ABB RobotStudio station: Celda_Robotica_Pintura_APM.rspag

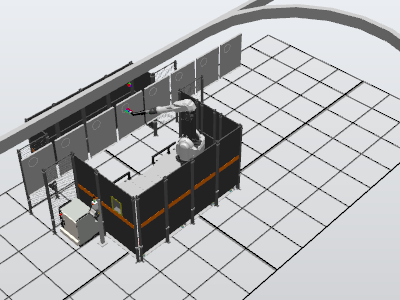
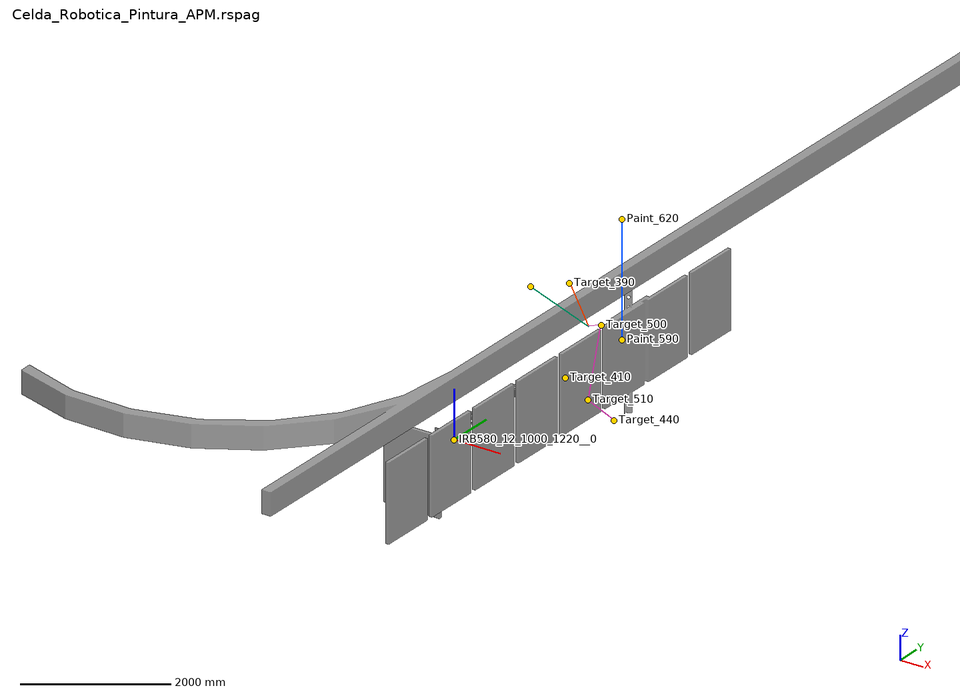
[picture v1: parts stored in the station drawn from their meshes, with robot base, taught points and paths (robot models come from the ABB library and are not in the file)]
--- station ---
Station Celda_Robotica_2_APM (saved by RobotStudio 23.3.10550.0)
Controller Controlador_Pintura_v2, task T_ROB1: task frame (RAPID world) sits at (2600, 704.38, 2665.12) mm, rotated rx 180 ry 0 rz 90 deg in the station
Controller Controlador_Pintura_v2
  mechanical unit ROB_1: IRB580_12_1000_1220__01, 6 joints, base frame (-1683.63, -1674.53, 2052.21) mm, rotated rx 180 ry 0 rz 0 deg
  mechanical unit CNV1: ?, 1 joints, base frame (-1079.32, 0, 0) mm
Layout (positions relative to the parent item):
  - Fence_800_AW [part, from Libraries\f3bba005-ce8c-4d92-bad9-ebedfeb7daa5fence_800_aw.rslib] at (-415.23, -1488.01, 0) mm
  - Pedestal_h440 [part, from Libraries\Pedestal_h440.rslib] at (891.47, -950, 628.29) mm, rotated rx 0 ry 0 rz 90 deg
  - sPallet250R_Single_rev1 [part, from Libraries\sPallet250R_Single_rev1.rslib] at (0, 1.5, 0) mm
  - ROBOBEL926_T_TD_03 [mechanism, from Libraries\ROBOBEL926_T_TD_03.rslib] at (1986.48, -515.02, 1892.16) mm, rotated rx -89.96 ry 0.02 rz -29.27 deg
  - Fence_800 [part, from Libraries\f3bba005-ce8c-4d92-bad9-ebedfeb7daa5fence_800_aw.rslib] at (-415.23, 1208.98, 0) mm
  - Fence_800_2 [part, from Libraries\f3bba005-ce8c-4d92-bad9-ebedfeb7daa5fence_800_aw.rslib] at (-415.23, -588.05, 0) mm
  - Fence_800_3 [part, from Libraries\f3bba005-ce8c-4d92-bad9-ebedfeb7daa5fence_800_aw.rslib] at (-415.23, 310.24, 0) mm
  - Fence_800_4 [part, from Libraries\f3bba005-ce8c-4d92-bad9-ebedfeb7daa5fence_800_aw.rslib] at (1805.95, -1488.01, 0) mm, rotated rx 0 ry 0 rz 90 deg
  - Fence_800_5 [part, from Libraries\f3bba005-ce8c-4d92-bad9-ebedfeb7daa5fence_800_aw.rslib] at (495.14, -1488.01, 0) mm, rotated rx 0 ry 0 rz 90 deg
  - Fence_800_6 [part, from Libraries\f3bba005-ce8c-4d92-bad9-ebedfeb7daa5fence_800_aw.rslib] at (1133.79, -1488.01, 0) mm, rotated rx 0 ry 0 rz 90 deg
  - Fence_800_7 [part, from Libraries\f3bba005-ce8c-4d92-bad9-ebedfeb7daa5fence_800_aw.rslib] at (2834.37, 2145.85, 0) mm, rotated rx 0 ry 0 rz -90 deg
  - IRC5_Singel-Cabinet [part, from Libraries\IRC5_Singel-Cabinet.rslib] at (1354.6, 2720.15, 100) mm, rotated rx 90 ry 0 rz 180 deg
  - Operator_panel [part, from Libraries\Operator_panel.rslib] at (714, 2359.02, 0) mm, rotated rx 0 ry 0 rz 90 deg
  - MeshModel_BoundingBox [graphiccomponentgroup]
  - MeshModel_ClippingPlane [graphiccomponentgroup]
  - MeshModel_ClippingCurve [graphiccomponentgroup]
  - Part5 [part], size 130 x 63 x 230 mm
  - Part6 [part], size 100 x 10 x 140 mm
  - Part7 [part], size 150 x 1 x 250 mm
  - Part8 [graphiccomponentgroup] at (0, 0, 420.53) mm
    - Part8_1 [part] at (2372.99, 892.19, 255.6) mm, rotated rx 90 ry 0 rz -151.74 deg, size 8 x 8 x 3 mm
    - Part8_2 [part] at (2372.99, 892.19, 255.6) mm, rotated rx 90 ry 0 rz -151.74 deg, size 8 x 8 x 3 mm
    - Part8_3 [part] at (2372.99, 892.19, 255.6) mm, rotated rx 90 ry 0 rz -151.74 deg, size 50 x 50 x 3 mm
    - Part8_4 [part] at (2372.99, 892.19, 255.6) mm, rotated rx 90 ry 0 rz -151.74 deg, size 8 x 8 x 3 mm
    - Part8_5 [part] at (2372.99, 892.19, 255.6) mm, rotated rx 90 ry 0 rz -151.74 deg, size 8 x 8 x 3 mm
    - Part8_6 [part] at (2372.99, 892.19, 255.6) mm, rotated rx 90 ry 0 rz -151.74 deg, size 50 x 50 x 3 mm
    - Part8_7 [part] at (2372.99, 892.19, 255.6) mm, rotated rx 90 ry 0 rz -151.74 deg, size 8 x 8 x 3 mm
    - Part8_8 [part] at (2372.99, 892.19, 255.6) mm, rotated rx 90 ry 0 rz -151.74 deg, size 50 x 50 x 3 mm
    - Part8_9 [part] at (2372.99, 892.19, 255.6) mm, rotated rx 90 ry 0 rz -151.74 deg, size 8 x 8 x 3 mm
    - Part8_10 [part] at (2372.99, 892.19, 255.6) mm, rotated rx 90 ry 0 rz -151.74 deg, size 50 x 50 x 3 mm
    - Part8_11 [part] at (2372.99, 892.19, 255.6) mm, rotated rx 90 ry 0 rz -151.74 deg, size 50 x 50 x 3 mm
    - Part8_12 [part] at (2372.99, 892.19, 255.6) mm, rotated rx 90 ry 0 rz -151.74 deg, size 8 x 8 x 3 mm
    - Part8_13 [part] at (2372.99, 892.19, 255.6) mm, rotated rx 90 ry 0 rz -151.74 deg, size 50 x 50 x 3 mm
    - Part8_14 [part] at (2372.99, 892.19, 255.6) mm, rotated rx 90 ry 0 rz -151.74 deg, size 50 x 50 x 3 mm
    - Part8_15 [part] at (2372.99, 892.19, 255.6) mm, rotated rx 90 ry 0 rz -151.74 deg, size 8 x 8 x 3 mm
    - Part8_16 [part] at (2372.99, 892.19, 255.6) mm, rotated rx 90 ry 0 rz -151.74 deg, size 50 x 50 x 3 mm
    - Part8_17 [part] at (2372.99, 892.19, 255.6) mm, rotated rx 90 ry 0 rz -151.74 deg, size 8 x 8 x 3 mm
    - Part8_18 [part] at (2372.99, 892.19, 255.6) mm, rotated rx 90 ry 0 rz -151.74 deg, size 50 x 50 x 3 mm
    - Part8_19 [part] at (2372.99, 892.19, 255.6) mm, rotated rx 90 ry 0 rz -151.74 deg, size 50 x 50 x 3 mm
    - Part8_20 [part] at (2372.99, 892.19, 255.6) mm, rotated rx 90 ry 0 rz -151.74 deg, size 8 x 8 x 3 mm
    - Part8_21 [part] at (2372.99, 892.19, 255.6) mm, rotated rx 90 ry 0 rz -151.74 deg, size 50 x 50 x 3 mm
    - Part8_22 [part] at (2372.99, 892.19, 255.6) mm, rotated rx 90 ry 0 rz -151.74 deg, size 50 x 50 x 3 mm
    - Part8_23 [part] at (2372.99, 892.19, 255.6) mm, rotated rx 90 ry 0 rz -151.74 deg, size 50 x 50 x 3 mm
    - Part8_24 [part] at (2372.99, 892.19, 255.6) mm, rotated rx 90 ry 0 rz -151.74 deg, size 8 x 8 x 3 mm
    - Part8_25 [part] at (2372.99, 892.19, 255.6) mm, rotated rx 90 ry 0 rz -151.74 deg, size 8 x 8 x 3 mm
    - Part8_26 [part] at (2372.99, 892.19, 255.6) mm, rotated rx 90 ry 0 rz -151.74 deg, size 50 x 50 x 3 mm
    - Part8_27 [part] at (2372.99, 892.19, 255.6) mm, rotated rx 90 ry 0 rz -151.74 deg, size 8 x 8 x 3 mm
    - Part8_28 [part] at (2372.99, 892.19, 255.6) mm, rotated rx 90 ry 0 rz -151.74 deg, size 8 x 8 x 3 mm
    - Part8_29 [part] at (2372.99, 892.19, 255.6) mm, rotated rx 90 ry 0 rz -151.74 deg, size 50 x 50 x 3 mm
    - Part8_30 [part] at (2372.99, 892.19, 255.6) mm, rotated rx 90 ry 0 rz -151.74 deg, size 8 x 8 x 3 mm
    - Part8_31 [part] at (2372.99, 892.19, 255.6) mm, rotated rx 90 ry 0 rz -151.74 deg, size 3 x 8 x 8 mm
    - Part8_32 [part] at (2372.99, 892.19, 255.6) mm, rotated rx 90 ry 0 rz -151.74 deg, size 3 x 8 x 8 mm
    - Part8_33 [part] at (2372.99, 892.19, 255.6) mm, rotated rx 90 ry 0 rz -151.74 deg, size 3 x 50 x 50 mm
    - Part8_34 [part] at (2372.99, 892.19, 255.6) mm, rotated rx 90 ry 0 rz -151.74 deg, size 3 x 8 x 8 mm
    - Part8_35 [part] at (2372.99, 892.19, 255.6) mm, rotated rx 90 ry 0 rz -151.74 deg, size 3 x 8 x 8 mm
    - Part8_36 [part] at (2372.99, 892.19, 255.6) mm, rotated rx 90 ry 0 rz -151.74 deg, size 3 x 50 x 50 mm
    - Part8_37 [part] at (2372.99, 892.19, 255.6) mm, rotated rx 90 ry 0 rz -151.74 deg, size 3 x 8 x 8 mm
    - Part8_38 [part] at (2372.99, 892.19, 255.6) mm, rotated rx 90 ry 0 rz -151.74 deg, size 3 x 50 x 50 mm
    - Part8_39 [part] at (2372.99, 892.19, 255.6) mm, rotated rx 90 ry 0 rz -151.74 deg, size 3 x 8 x 8 mm
    - Part8_40 [part] at (2372.99, 892.19, 255.6) mm, rotated rx 90 ry 0 rz -151.74 deg, size 3 x 50 x 50 mm
    - Part8_41 [part] at (2372.99, 892.19, 255.6) mm, rotated rx 90 ry 0 rz -151.74 deg, size 3 x 50 x 50 mm
    - Part8_42 [part] at (2372.99, 892.19, 255.6) mm, rotated rx 90 ry 0 rz -151.74 deg, size 3 x 8 x 8 mm
    - Part8_43 [part] at (2372.99, 892.19, 255.6) mm, rotated rx 90 ry 0 rz -151.74 deg, size 3 x 50 x 50 mm
    - Part8_44 [part] at (2372.99, 892.19, 255.6) mm, rotated rx 90 ry 0 rz -151.74 deg, size 3 x 50 x 50 mm
    - Part8_45 [part] at (2372.99, 892.19, 255.6) mm, rotated rx 90 ry 0 rz -151.74 deg, size 3 x 8 x 8 mm
    - Part8_46 [part] at (2372.99, 892.19, 255.6) mm, rotated rx 90 ry 0 rz -151.74 deg, size 3 x 50 x 50 mm
    - Part8_47 [part] at (2372.99, 892.19, 255.6) mm, rotated rx 90 ry 0 rz -151.74 deg, size 3 x 8 x 8 mm
    - Part8_48 [part] at (2372.99, 892.19, 255.6) mm, rotated rx 90 ry 0 rz -151.74 deg, size 3 x 50 x 50 mm
    - Part8_49 [part] at (2372.99, 892.19, 255.6) mm, rotated rx 90 ry 0 rz -151.74 deg, size 3 x 50 x 50 mm
    - Part8_50 [part] at (2372.99, 892.19, 255.6) mm, rotated rx 90 ry 0 rz -151.74 deg, size 3 x 8 x 8 mm
    - Part8_51 [part] at (2372.99, 892.19, 255.6) mm, rotated rx 90 ry 0 rz -151.74 deg, size 3 x 50 x 50 mm
    - Part8_52 [part] at (2372.99, 892.19, 255.6) mm, rotated rx 90 ry 0 rz -151.74 deg, size 3 x 50 x 50 mm
    - Part8_53 [part] at (2372.99, 892.19, 255.6) mm, rotated rx 90 ry 0 rz -151.74 deg, size 3 x 50 x 50 mm
    - Part8_54 [part] at (2372.99, 892.19, 255.6) mm, rotated rx 90 ry 0 rz -151.74 deg, size 3 x 8 x 8 mm
    - Part8_55 [part] at (2372.99, 892.19, 255.6) mm, rotated rx 90 ry 0 rz -151.74 deg, size 3 x 8 x 8 mm
    - Part8_56 [part] at (2372.99, 892.19, 255.6) mm, rotated rx 90 ry 0 rz -151.74 deg, size 3 x 50 x 50 mm
    - Part8_57 [part] at (2372.99, 892.19, 255.6) mm, rotated rx 90 ry 0 rz -151.74 deg, size 3 x 8 x 8 mm
    - Part8_58 [part] at (2372.99, 892.19, 255.6) mm, rotated rx 90 ry 0 rz -151.74 deg, size 3 x 8 x 8 mm
    - Part8_59 [part] at (2372.99, 892.19, 255.6) mm, rotated rx 90 ry 0 rz -151.74 deg, size 3 x 50 x 50 mm
    - Part8_60 [part] at (2372.99, 892.19, 255.6) mm, rotated rx 90 ry 0 rz -151.74 deg, size 3 x 8 x 8 mm
    - Part8_61 [part] at (2372.99, 892.19, 255.6) mm, rotated rx 90 ry 0 rz -151.74 deg, size 100 x 2000 x 0 mm
    - Part8_62 [part] at (2372.99, 892.19, 255.6) mm, rotated rx 90 ry 0 rz -151.74 deg, size 0 x 2000 x 3 mm
    - Part8_63 [part] at (2372.99, 892.19, 255.6) mm, rotated rx 90 ry 0 rz -151.74 deg, size 97 x 2000 x 0 mm
    - Part8_64 [part] at (2372.99, 892.19, 255.6) mm, rotated rx 90 ry 0 rz -151.74 deg, size 0 x 2000 x 97 mm
    - Part8_65 [part] at (2372.99, 892.19, 255.6) mm, rotated rx 90 ry 0 rz -151.74 deg, size 3 x 2000 x 0 mm
    - Part8_66 [part] at (2372.99, 892.19, 255.6) mm, rotated rx 90 ry 0 rz -151.74 deg, size 0 x 2000 x 100 mm
    - Part8_67 [part] at (2372.99, 892.19, 255.6) mm, rotated rx 90 ry 0 rz -151.74 deg, size 100 x 0 x 100 mm
    - Part8_68 [part] at (2372.99, 892.19, 255.6) mm, rotated rx 90 ry 0 rz -151.74 deg, size 100 x 0 x 100 mm
  - Fence_800_8 [part, from Libraries\f3bba005-ce8c-4d92-bad9-ebedfeb7daa5fence_800_aw.rslib] at (927.36, 2145.85, 0) mm, rotated rx 0 ry 0 rz -90 deg
  - Fence_800_9 [part, from Libraries\f3bba005-ce8c-4d92-bad9-ebedfeb7daa5fence_800_aw.rslib] at (3699.9, 2145.85, 0) mm, rotated rx 0 ry 0 rz 180 deg
  - Fence_1200_AW [part, from Libraries\48bacffd-50a7-42ca-88af-306811f71c63fence_1200_aw_ts.rslib] at (-372.93, 2145.84, -3.07) mm, rotated rx 0 ry 0 rz -90 deg
  - Fence_800_10 [part, from Libraries\f3bba005-ce8c-4d92-bad9-ebedfeb7daa5fence_800_aw.rslib] at (3699.9, 1245.66, 0) mm, rotated rx 0 ry 0 rz 180 deg
  - Fence_800_11 [part, from Libraries\f3bba005-ce8c-4d92-bad9-ebedfeb7daa5fence_800_aw.rslib] at (3699.9, 346.45, 0) mm, rotated rx 0 ry 0 rz 180 deg
  - Fence_800_12 [part, from Libraries\f3bba005-ce8c-4d92-bad9-ebedfeb7daa5fence_800_aw.rslib] at (3699.9, -552.32, 0) mm, rotated rx 0 ry 0 rz 180 deg
  - Fence_800_13 [part, from Libraries\f3bba005-ce8c-4d92-bad9-ebedfeb7daa5fence_800_aw.rslib] at (3709.4, -1462.88, 0) mm, rotated rx 0 ry 0 rz 90 deg
  - Troax_800_Poles [part, from Libraries\9d9a1cc8-97d7-4a8c-92c3-0b58d3e22f0ctroax_800_poles.rslib] at (1795.44, -1936.07, 0) mm
  - Troax_800 [part, from Libraries\9d9a1cc8-97d7-4a8c-92c3-0b58d3e22f0ctroax_800_poles.rslib] at (2844.71, -1936.07, 0) mm
  - Troax_801 [part, from Libraries\9d9a1cc8-97d7-4a8c-92c3-0b58d3e22f0ctroax_800_poles.rslib] at (2844.71, 2565.66, 0) mm
  - Troax_802 [part, from Libraries\9d9a1cc8-97d7-4a8c-92c3-0b58d3e22f0ctroax_800_poles.rslib] at (1839.74, 2565.66, 0) mm
  - IRB580_12_1000_1220__01 [mechanism, from Libraries\IRB580_12_1000_1220_G_01.rslib] at (925.47, -979.26, 612.91) mm, rotated rx 0 ry 0 rz 90 deg; joint values [-1.2473, 0.0041, 0.4831, 0.7898, -0.7583, -2.5492] (rad or m)
  - SC_SprayFans [graphiccomponentgroup]
  - Conveyor [conveyor]
    - Part1 [part] at (425.3, 1739.05, 2665.12) mm, rotated rx 90 ry 0 rz 0 deg, size 4829.7 x 351 x 20000 mm
    - Part12 [part], size 900 x 53 x 1200 mm
    - ConveyorObject_142 [conveyorobject] at (2600, 2959.94, 2665.12) mm, rotated rx 180 ry 0 rz 90 deg
      - Part12 [part] at (200, -100, 450) mm, rotated rx 180 ry 0 rz 0 deg, size 900 x 53 x 1200 mm
    - ConveyorObject_143 [conveyorobject] at (2600, 1959.94, 2665.12) mm, rotated rx 180 ry 0 rz 90 deg
      - Part12 [part] at (200, -100, 450) mm, rotated rx 180 ry 0 rz 0 deg, size 900 x 53 x 1200 mm
    - ConveyorObject_144 [conveyorobject] at (2600, 959.94, 2665.12) mm, rotated rx 180 ry 0 rz 90 deg
      - Part12 [part] at (200, -100, 450) mm, rotated rx 180 ry 0 rz 0 deg, size 900 x 53 x 1200 mm
    - ConveyorObject_13 [conveyorobject] at (2600, -40.06, 2665.12) mm, rotated rx 180 ry 0 rz 90 deg
      - Part12 [part] at (200, -100, 450) mm, rotated rx 180 ry 0 rz 0 deg, size 900 x 53 x 1200 mm
    - ConveyorObject_14 [conveyorobject] at (2600, -1040.06, 2665.12) mm, rotated rx 180 ry 0 rz 90 deg
      - Part12 [part] at (200, -100, 450) mm, rotated rx 180 ry 0 rz 0 deg, size 900 x 53 x 1200 mm
    - ConveyorObject_15 [conveyorobject] at (2600, -2040.06, 2665.12) mm, rotated rx 180 ry 0 rz 90 deg
      - Part12 [part] at (200, -100, 450) mm, rotated rx 180 ry 0 rz 0 deg, size 900 x 53 x 1200 mm
    - ConveyorObject_16 [conveyorobject] at (2600, -3040.06, 2665.12) mm, rotated rx 180 ry 0 rz 90 deg
      - Part12 [part] at (200, -100, 450) mm, rotated rx 180 ry 0 rz 0 deg, size 900 x 53 x 1200 mm
    - ConveyorObject_17 [conveyorobject] at (2600, -4040.06, 2665.12) mm, rotated rx 180 ry 0 rz 90 deg
      - Part12 [part] at (200, -100, 450) mm, rotated rx 180 ry 0 rz 0 deg, size 900 x 53 x 1200 mm
  - Part12 [graphiccomponentgroup] at (2486.98, -1946.56, 0) mm, rotated rx 0 ry 0 rz 90.74 deg
    - Part12_1 [part] at (3303.04, 0, 2213.48) mm, size 8 x 8 x 3 mm
    - Part12_2 [part] at (3303.04, 0, 2213.48) mm, size 8 x 8 x 3 mm
    - Part12_3 [part] at (3303.04, 0, 2213.48) mm, size 0 x 50 x 1194 mm
    - Part12_4 [part] at (3303.04, 0, 2213.48) mm, size 894 x 50 x 0 mm
    - Part12_5 [part] at (3303.04, 0, 2213.48) mm, size 0 x 50 x 1194 mm
    - Part12_6 [part] at (3303.04, 0, 2213.48) mm, size 894 x 50 x 0 mm
    - Part12_7 [part] at (3303.04, 0, 2213.48) mm, size 900 x 0 x 1200 mm
    - Part12_8 [part] at (3303.04, 0, 2213.48) mm, size 0 x 53 x 1200 mm
    - Part12_9 [part] at (3303.04, 0, 2213.48) mm, size 900 x 53 x 0 mm
    - Part12_10 [part] at (3303.04, 0, 2213.48) mm, size 0 x 53 x 1200 mm
    - Part12_11 [part] at (3303.04, 0, 2213.48) mm, size 900 x 53 x 0 mm
    - Part12_12 [part] at (3303.04, 0, 2213.48) mm, size 894 x 0 x 1194 mm
    - Part12_13 [part] at (3303.04, 0, 2213.48) mm, size 900 x 0 x 1200 mm
  - Part8 [part], size 100 x 2000 x 100 mm
Attachment: ROBOBEL926_T_TD_03 is attached to IRB580_12_1000_1220__01 / Link6
Attachment: Pedestal_h440 is attached to IRB580_12_1000_1220__01 / Base
Conveyor tracking Connection: unit CNV1, TravelOffset=4.2, QueueTrackDistance=0, StartWindowWidth=1.5, SyncSeparation=0.1, CountsPerMeter=10000
Targets, tools, work objects and paths stored in the station and not in the controller backup, written as RAPID:
! task T_ROB1
MODULE m4
  PROC Path_10()
    SetBrush 3\Z:=-119.15;
    SetBrush 3\Z:=-1042.15;
    SetBrush 3\Z:=-1046.00;
    SetBrush 3\Z:=-154.00;
    SetBrush 3\Z:=-154.00;
    SetBrush 3\Z:=-1046.00;
    SetBrush 3\Z:=-1046.00;
    SetBrush 3\Z:=-154.00;
    SetBrush 3\Z:=-154.00;
    SetBrush 3\Z:=-1046.00;
    SetBrush 3\Z:=-1046.00;
    SetBrush 1\Z:=97.00;
  ENDPROC
ENDMODULE


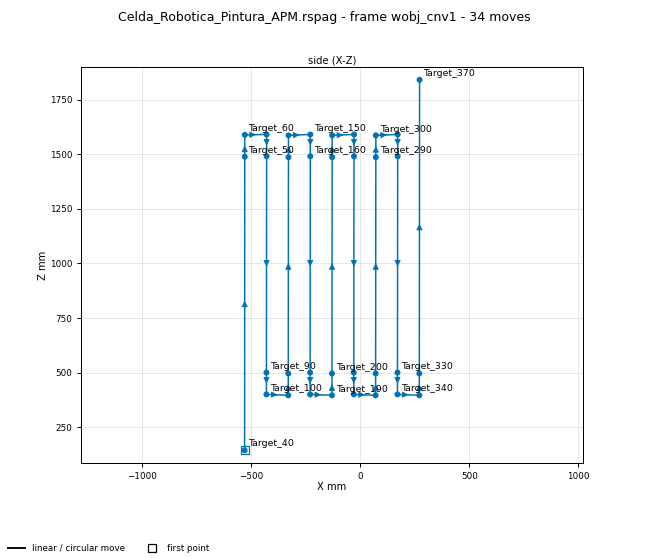
[picture p0: tool path of Celda_Robotica_Pintura_APM.rspag in frame wobj_cnv1, 34 of 52 moves have a stored position in this frame; points joined in program order, loops and branches not executed]
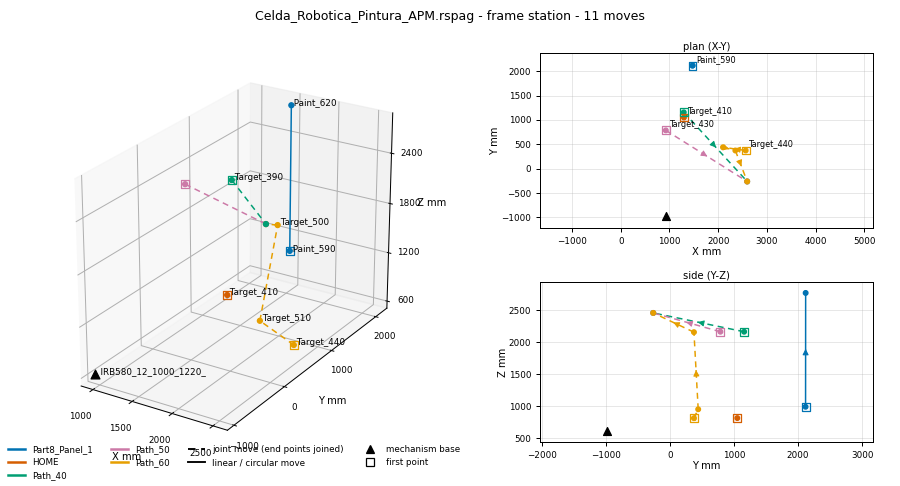
[picture p1: tool path of Celda_Robotica_Pintura_APM.rspag in frame station, 11 of 52 moves have a stored position in this frame; points joined in program order, loops and branches not executed]
--- Backups/Controlador_Pintura_v2/RAPID/TASK0/SYSMOD/userlog.sys ---
module userlog(sysmodule)



   local const num MAX_LOG_SIZE   := 100000; ! Size in bytes.
   local const num MAX_LOG_FILES  := 5;
   local const num MAX_LOG_BUFFER := 20; ! Entries to keep before flushing.



   ! Keep persistent to survive restarts and share between tasks.
   pers string stUserLogBuffer{MAX_LOG_BUFFER};
   pers string stUserLogTime{MAX_LOG_BUFFER};
   pers num nUserLogIndex;
   pers num nUserLogFileNo;

   pers bool bUserBufAddSem;
   pers bool bUserFlushSem;



   proc PntUserLog(string stMessage \Switch Flush)
      BufferAdd stMessage;
      if Present(Flush)
         FlushBuffer;
   endproc



   local proc BufferAdd(string stMessage)
      var bool bTimeOut;

      WaitUntil TestAndSet(bUserBufAddSem) \MaxTime := 1 \TimeFlag := bTimeOut;
      if bTimeOut then
         ErrWrite "PntUserLog Error", "Buffer Add Semaphore Timeout";
         bUserBufAddSem := false; ! Force release.
         return;
      endif

      stUserLogBuffer{nUserLogIndex} := stMessage;
      stUserLogTime{nUserLogIndex} := CDate() + " " + CTime();

      Incr nUserLogIndex;
      if nUserLogIndex > MAX_LOG_BUFFER then
         ! Must be flushed.
         FlushBuffer;
      endif

      bUserBufAddSem := false; ! Release.
   error
      if errno = ERR_OUTOFBND then
         Decr nUserLogIndex;
         retry;
      endif
   endproc



   local proc FlushBuffer()
      var bool bTimeOut;
      var iodev ioLog;
      var string stLogFile;

      WaitUntil TestAndSet(bUserFlushSem) \MaxTime := 1 \TimeFlag := bTimeOut;
      if bTimeOut then
         ErrWrite "PntUserLog Error", "Flush Semaphore Timeout";
         bUserFlushSem := false; ! Force release.
         return;
      endif

      if nUserLogIndex <= 1 then
         bUserFlushSem := false;
         return; ! Buffer empty, nothing to flush.
      endif

      stLogFile := "HOME:/logs/user" + ValToStr(nUserLogFileNo) + ".log";

      Open stLogFile, ioLog \Append;
      for i from 1 to nUserLogIndex - 1 do ! Will normally be incremented to one above.
         Write ioLog, stUserLogTime{i} + " " \NoNewLine;
         Write ioLog, stUserLogBuffer{i};
      endfor
      Close ioLog;
      nUserLogIndex := 1;

      if FileSize(stLogFile) > MAX_LOG_SIZE then
         Incr nUserLogFileNo;
         if nUserLogFileNo > MAX_LOG_FILES
            nUserLogFileNo := 1;

         stLogFile := "HOME:/logs/user" + ValToStr(nUserLogFileNo) + ".log";
         Open stLogFile, ioLog;
         Close ioLog;
      endif

      bUserFlushSem := false;
   error
      nUserLogIndex := 1;
      bUserFlushSem := false;
      return;
   endproc



   proc InitUserLog()
      bUserBufAddSem := false;
      bUserFlushSem := false;
      if nUserLogIndex = 0
         nUserLogIndex := 1;
      if nUserLogFileNo = 0
         nUserLogFileNo := 1;
   endproc



endmodule

--- Backups/Controlador_Pintura_v2/RAPID/TASK1/PROGMOD/CalibData.mod ---
MODULE CalibData
    PERS tooldata ROBOBEL926_T_TD_0:=[TRUE,[[117,0,470],[0.866025404,0,0.5,0]],[5.5,[30,0,225],[1,0,0,0],0,0,0]];
    PERS tooldata ROBOBEL926_T_TD_100:=[TRUE,[[204,0,520],[0.866025404,0,0.5,0]],[5.5,[30,0,225],[1,0,0,0],0,0,0]];
    PERS tooldata ROBOBEL926_T_TD_120:=[TRUE,[[220,0,530],[0.866025404,0,0.5,0]],[5.5,[30,0,225],[1,0,0,0],0,0,0]];
    PERS tooldata ROBOBEL926_T_TD_150:=[TRUE,[[247,0,545],[0.866025404,0,0.5,0]],[5.5,[30,0,225],[1,0,0,0],0,0,0]];
    PERS tooldata ROBOBEL926_T_TD_200:=[TRUE,[[290,0,570],[0.866025404,0,0.5,0]],[5.5,[30,0,225],[1,0,0,0],0,0,0]];
    PERS tooldata ROBOBEL926_T_TD_250:=[TRUE,[[333,0,595],[0.866025404,0,0.5,0]],[5.5,[30,0,225],[1,0,0,0],0,0,0]];
    PERS tooldata ROBOBEL926_T_TD_300:=[TRUE,[[377,0,620],[0.866025404,0,0.5,0]],[5.5,[30,0,225],[1,0,0,0],0,0,0]];
    TASK PERS wobjdata Workobject_x:=[FALSE,TRUE,"",[[-1312.950919555,-1305.931066272,2052.209095741],[0,1,0,0]],[[0,0,0],[1,0,0,0]]];
    TASK PERS wobjdata Workobject_2:=[FALSE,TRUE,"",[[304.880323441,-1115.931066272,2052.444095741],[0,1,0,0]],[[0,0,0],[1,0,0,0]]];
    TASK PERS wobjdata Workobject_Y:=[FALSE,TRUE,"",[[-1033.633323441,-1305.931066272,2052.209095741],[0,1,0,0]],[[0,0,0],[1,0,0,0]]];
    TASK PERS wobjdata wobj_cnv1:=[FALSE,FALSE,"CNV1",[[0,0,0],[1,0,0,0]],[[0,0,0],[1,0,0,0]]];
ENDMODULE

--- Backups/Controlador_Pintura_v2/RAPID/TASK1/PROGMOD/m4.mod ---
MODULE m4
    LOCAL CONST robtarget Paint_590:=[[1107.577696927,10.451886223,381.900082634],[0.171778362,0.171777942,0.68592355,0.685925227],[0,0,0,0],[9E+09,9E+09,9E+09,9E+09,9E+09,9E+09]];
    LOCAL CONST robtarget Paint_620:=[[1108.897947742,9.717576103,2159.750024363],[0.185869223,0.185876599,0.682253423,0.682226348],[0,0,0,0],[9E+09,9E+09,9E+09,9E+09,9E+09,9E+09]];
    PROC Part8_Panel_1()
        ActUnit CNV1;
        ConfL\Off;
        PaintL Paint_590,v800,z100,ROBOBEL926_T_TD_120\WObj:=Workobject_2;
        SetBrush 3\Z:=-880.03;
        PaintL Paint_620,v800,z100,ROBOBEL926_T_TD_120\WObj:=Workobject_2;
    ENDPROC
ENDMODULE

--- Backups/Controlador_Pintura_v2/RAPID/TASK1/PROGMOD/Module1.mod ---
MODULE Module1
    CONST robtarget Target_10:=[[1840.7,0,1423.5],[0.258819045,0,0.965925826,0],[0,0,-1,0],[9E+09,9E+09,9E+09,9E+09,9E+09,0]];
    CONST robtarget Target_20:=[[892.866653856,-1609.654111301,1423.52749384],[0.225824589,0.49248749,0.830925505,-0.126578561],[-1,2,-3,0],[9E+09,9E+09,9E+09,9E+09,9E+09,0]];
    CONST robtarget Target_30:=[[740.142294984,-1332.710931703,577.907289687],[0.016121954,0.510934614,0.859461686,-0.003392987],[-1,2,-3,0],[9E+09,9E+09,9E+09,9E+09,9E+09,0]];
    CONST robtarget Target_40:=[[-528.272188377,27.479862138,144.772889571],[0.005341212,0.005394694,0.707059088,0.707113721],[-1,1,1,0],[9E+09,9E+09,9E+09,9E+09,9E+09,0]];
    CONST robtarget Target_50:=[[-527.572745869,23.353740717,1488.539132077],[0.004074075,0.004796881,0.706974183,0.707211352],[-1,2,0,0],[9E+09,9E+09,9E+09,9E+09,9E+09,0]];
    CONST robtarget Target_60:=[[-527.488942032,23.325481167,1588.516095022],[0.004074322,0.004781672,0.706973503,0.707212133],[-1,2,0,0],[9E+09,9E+09,9E+09,9E+09,9E+09,0]];
    CONST robtarget Target_70:=[[-427.487838107,22.05305561,1590.525193202],[0.004074556,0.004787048,0.706973257,0.707212342],[-1,2,0,0],[9E+09,9E+09,9E+09,9E+09,9E+09,0]];
    CONST robtarget Target_80:=[[-427.572393813,22.080226384,1490.543554698],[0.004074275,0.004801879,0.706975355,0.707210145],[-1,2,0,0],[9E+09,9E+09,9E+09,9E+09,9E+09,0]];
    CONST robtarget Target_90:=[[-428.39747985,22.362471871,500.408170806],[0.004142759,0.004896114,0.70704969,0.707134783],[-1,2,0,0],[9E+09,9E+09,9E+09,9E+09,9E+09,0]];
    CONST robtarget Target_100:=[[-428.492137513,22.373047089,400.38407293],[0.004147301,0.004897982,0.707057999,0.707126435],[-1,2,0,0],[9E+09,9E+09,9E+09,9E+09,9E+09,0]];
    CONST robtarget Target_110:=[[-328.494793387,21.099793583,396.363555684],[0.004155071,0.00489719,0.707061405,0.707122989],[-1,2,0,0],[9E+09,9E+09,9E+09,9E+09,9E+09,0]];
    CONST robtarget Target_120:=[[-328.399866869,21.089122834,496.391143398],[0.00415027,0.004895925,0.707051642,0.707132788],[-1,2,0,0],[9E+09,9E+09,9E+09,9E+09,9E+09,0]];
    CONST robtarget Target_130:=[[-327.56763526,20.819515861,1486.546476442],[0.004079524,0.004810491,0.706975784,0.707209627],[-1,2,0,0],[9E+09,9E+09,9E+09,9E+09,9E+09,0]];
    CONST robtarget Target_140:=[[-327.486669583,20.788362511,1586.532424361],[0.004077363,0.004795023,0.706973187,0.707212341],[-1,2,0,0],[9E+09,9E+09,9E+09,9E+09,9E+09,0]];
    CONST robtarget Target_150:=[[-227.479008283,19.521465484,1590.538488911],[0.00408025,0.004801621,0.706973034,0.707212433],[-1,2,0,0],[9E+09,9E+09,9E+09,9E+09,9E+09,0]];
    CONST robtarget Target_160:=[[-227.561626585,19.550554509,1490.548324827],[0.004082953,0.004815363,0.706975989,0.70720937],[-1,2,0,0],[9E+09,9E+09,9E+09,9E+09,9E+09,0]];
    CONST robtarget Target_170:=[[-228.396815796,19.813031972,500.383493147],[0.004155351,0.004896299,0.707052247,0.707132151],[-1,2,0,0],[9E+09,9E+09,9E+09,9E+09,9E+09,0]];
    CONST robtarget Target_180:=[[-228.491534337,19.823567274,400.351761225],[0.004160481,0.00489727,0.707063163,0.7071212],[-1,2,0,0],[9E+09,9E+09,9E+09,9E+09,9E+09,0]];
    CONST robtarget Target_190:=[[-128.497212182,18.546806917,396.342313584],[0.004164662,0.004898105,0.707065032,0.7071193],[-1,2,0,0],[9E+09,9E+09,9E+09,9E+09,9E+09,0]];
    CONST robtarget Target_200:=[[-128.402283376,18.537773943,496.374601764],[0.00415957,0.004897287,0.707053506,0.707130861],[-1,2,0,0],[9E+09,9E+09,9E+09,9E+09,9E+09,0]];
    CONST robtarget Target_210:=[[-127.559686337,18.287720725,1486.547459841],[0.004088326,0.004821514,0.706976397,0.707208889],[-1,2,0,0],[9E+09,9E+09,9E+09,9E+09,9E+09,0]];
    CONST robtarget Target_220:=[[-127.475861123,18.260698663,1586.542508113],[0.004083964,0.004810572,0.706974288,0.707211097],[-1,2,0,0],[9E+09,9E+09,9E+09,9E+09,9E+09,0]];
    CONST robtarget Target_230:=[[-27.465275948,16.99772691,1590.543846301],[0.004089307,0.004817332,0.706974697,0.707210612],[-1,2,0,0],[9E+09,9E+09,9E+09,9E+09,9E+09,0]];
    CONST robtarget Target_240:=[[-27.549996265,17.023405636,1490.546068498],[0.00409402,0.004827299,0.706977098,0.707208116],[-1,2,0,0],[9E+09,9E+09,9E+09,9E+09,9E+09,0]];
    CONST robtarget Target_250:=[[-28.401181507,17.260029965,500.372144944],[0.004162476,0.0048984,0.7070536,0.707130742],[-1,2,0,0],[9E+09,9E+09,9E+09,9E+09,9E+09,0]];
    CONST robtarget Target_260:=[[-28.496140656,17.269016618,400.338123467],[0.004167521,0.004899351,0.707065754,0.707118553],[-1,2,0,0],[9E+09,9E+09,9E+09,9E+09,9E+09,0]];
    CONST robtarget Target_270:=[[71.49679788,15.992206778,396.332227298],[0.00417006,0.004900903,0.707067504,0.707116778],[-1,3,-1,0],[9E+09,9E+09,9E+09,9E+09,9E+09,0]];
    CONST robtarget Target_280:=[[71.592483669,15.983145712,496.363299783],[0.004165681,0.004899913,0.707055858,0.707128455],[-1,3,-1,0],[9E+09,9E+09,9E+09,9E+09,9E+09,0]];
    CONST robtarget Target_290:=[[72.455283813,15.765018327,1486.540739891],[0.004102274,0.004834318,0.706978132,0.707206987],[-1,2,0,0],[9E+09,9E+09,9E+09,9E+09,9E+09,0]];
    CONST robtarget Target_300:=[[72.54192036,15.740748378,1586.541200077],[0.004097317,0.004825394,0.706975437,0.70720977],[-1,2,0,0],[9E+09,9E+09,9E+09,9E+09,9E+09,0]];
    CONST robtarget Target_310:=[[172.553508551,14.479398174,1590.540711743],[0.004102491,0.004833384,0.70697748,0.707207643],[-1,2,0,0],[9E+09,9E+09,9E+09,9E+09,9E+09,0]];
    CONST robtarget Target_320:=[[172.466869062,14.50197769,1490.538176011],[0.004107506,0.004841425,0.706980449,0.707204591],[-1,2,0,0],[9E+09,9E+09,9E+09,9E+09,9E+09,0]];
    CONST robtarget Target_330:=[[171.593230938,14.705288225,500.359164806],[0.004168079,0.004901497,0.707057346,0.707126942],[-1,3,-1,0],[9E+09,9E+09,9E+09,9E+09,9E+09,0]];
    CONST robtarget Target_340:=[[171.496956558,14.713624894,400.32946553],[0.004171779,0.00490269,0.707068588,0.70711567],[-1,3,-1,0],[9E+09,9E+09,9E+09,9E+09,9E+09,0]];
    CONST robtarget Target_350:=[[271.489204751,13.435299841,396.324988838],[0.00417321,0.004904865,0.707070721,0.707113514],[-1,3,-1,0],[9E+09,9E+09,9E+09,9E+09,9E+09,0]];
    CONST robtarget Target_360:=[[271.586482838,13.429144646,496.350016771],[0.004170558,0.00490345,0.70706039,0.70712387],[-1,3,-1,0],[9E+09,9E+09,9E+09,9E+09,9E+09,0]];
    CONST robtarget Target_370:=[[272.785926297,13.172503921,1840.539357733],[0.004098663,0.004824734,0.706974774,0.70721043],[-1,2,0,0],[9E+09,9E+09,9E+09,9E+09,9E+09,0]];
    CONST robtarget Target_380:=[[1871.516358775,-1298.822789134,1497.518343998],[0.00490345,-0.004170558,0.70712387,-0.70706039],[-1,3,-1,0],[9E+09,9E+09,9E+09,9E+09,9E+09,0]];
    CONST robtarget Target_400:=[[1071.556192092,-1299.116793612,1847.338710432],[0.005357911,-0.005363904,0.707079393,-0.707093525],[-1,0,-2,0],[9E+09,9E+09,9E+09,9E+09,9E+09,0]];
    CONST robtarget Target_410:=[[346.014287013,-1302.17449256,1847.3786284],[0.005307132,-0.005376763,0.70704125,-0.70713195],[-1,0,-2,0],[9E+09,9E+09,9E+09,9E+09,9E+09,0]];
    CONST robtarget Target_390:=[[1765.7,0,1553.5],[0.258819045,0,0.965925826,0],[-1,1,-2,0],[9E+09,9E+09,9E+09,9E+09,9E+09,0]];
    CONST robtarget Target_420:=[[871.479680582,-1302.22633464,1847.391793055],[0.005226588,-0.005399518,0.706991469,-0.707182149],[-1,0,-2,0],[9E+09,9E+09,9E+09,9E+09,9E+09,0]];
    CONST robtarget Target_430:=[[1395.017596114,368.598558674,1553.5],[0.258819045,0,0.965925826,0],[-1,0,-1,0],[9E+09,9E+09,9E+09,9E+09,9E+09,0]];
    CONST robtarget Target_440:=[[981.896827244,-1271.558575619,203.169081023],[0.031794427,0.009492169,0.735782467,-0.676404594],[-1,1,-3,0],[9E+09,9E+09,9E+09,9E+09,9E+09,0]];
    CONST robtarget Target_450:=[[1329.978948042,-989.38883415,884.448705644],[0.031699125,0.00901064,0.735631304,-0.676580046],[-1,1,-3,0],[9E+09,9E+09,9E+09,9E+09,9E+09,0]];
    CONST robtarget Target_460:=[[1330.135466443,-373.807440649,884.445594571],[0.031688949,0.008760507,0.735500141,-0.67672639],[-1,1,-3,0],[9E+09,9E+09,9E+09,9E+09,9E+09,0]];
    CONST robtarget Target_470:=[[1330.166917335,-373.770492946,1530.203031462],[0.03168344,0.008713699,0.735460486,-0.676770349],[-1,1,-3,0],[9E+09,9E+09,9E+09,9E+09,9E+09,0]];
    CONST robtarget Target_480:=[[205.079487849,-1271.520713426,1435.697333288],[0.031553283,0.009171046,0.735654959,-0.676558987],[-1,0,-2,0],[9E+09,9E+09,9E+09,9E+09,9E+09,0]];
    CONST robtarget Target_490:=[[1046.332947544,-985.816330668,1598.37529885],[0.018422806,0.002718833,0.721287549,-0.692385355],[-1,0,-2,0],[9E+09,9E+09,9E+09,9E+09,9E+09,0]];
    CONST robtarget Target_510:=[[1048.360884478,-805.975935616,342.427266896],[0.051245728,-0.005471976,0.740865703,-0.669673012],[-1,1,-3,0],[9E+09,9E+09,9E+09,9E+09,9E+09,0]];
    CONST robtarget Target_500:=[[981.922888278,-1059.580450522,1546.689786441],[0.031649674,0.009245031,0.73566951,-0.676537656],[-1,0,-2,0],[9E+09,9E+09,9E+09,9E+09,9E+09,0]];
    PROC Path_20()
        MoveL Target_40,v1500,z100,ROBOBEL926_T_TD_300\WObj:=wobj_cnv1;MoveL Target_50,v1500,z100,ROBOBEL926_T_TD_300\WObj:=wobj_cnv1;
        MoveL Target_60,v1500,z100,ROBOBEL926_T_TD_300\WObj:=wobj_cnv1;
        MoveL Target_70,v1500,z100,ROBOBEL926_T_TD_300\WObj:=wobj_cnv1;
        MoveL Target_80,v1500,z100,ROBOBEL926_T_TD_300\WObj:=wobj_cnv1;
        MoveL Target_90,v1500,z100,ROBOBEL926_T_TD_300\WObj:=wobj_cnv1;
        MoveL Target_100,v1500,z100,ROBOBEL926_T_TD_300\WObj:=wobj_cnv1;
        MoveL Target_110,v1500,z100,ROBOBEL926_T_TD_300\WObj:=wobj_cnv1;
        MoveL Target_120,v1500,z100,ROBOBEL926_T_TD_300\WObj:=wobj_cnv1;
        MoveL Target_130,v1500,z100,ROBOBEL926_T_TD_300\WObj:=wobj_cnv1;
        MoveL Target_140,v1500,z100,ROBOBEL926_T_TD_300\WObj:=wobj_cnv1;
        MoveL Target_150,v1500,z100,ROBOBEL926_T_TD_300\WObj:=wobj_cnv1;
        MoveL Target_160,v1500,z100,ROBOBEL926_T_TD_300\WObj:=wobj_cnv1;
        MoveL Target_170,v1500,z100,ROBOBEL926_T_TD_300\WObj:=wobj_cnv1;
        MoveL Target_180,v1500,z100,ROBOBEL926_T_TD_300\WObj:=wobj_cnv1;
        MoveL Target_190,v1500,z100,ROBOBEL926_T_TD_300\WObj:=wobj_cnv1;
        MoveL Target_200,v1500,z100,ROBOBEL926_T_TD_300\WObj:=wobj_cnv1;
        MoveL Target_210,v1500,z100,ROBOBEL926_T_TD_300\WObj:=wobj_cnv1;
        MoveL Target_220,v1500,z100,ROBOBEL926_T_TD_300\WObj:=wobj_cnv1;
        MoveL Target_230,v1500,z100,ROBOBEL926_T_TD_300\WObj:=wobj_cnv1;
        MoveL Target_240,v1500,z100,ROBOBEL926_T_TD_300\WObj:=wobj_cnv1;
        MoveL Target_250,v1500,z100,ROBOBEL926_T_TD_300\WObj:=wobj_cnv1;
        MoveL Target_260,v1500,z100,ROBOBEL926_T_TD_300\WObj:=wobj_cnv1;
        MoveL Target_270,v1500,z100,ROBOBEL926_T_TD_300\WObj:=wobj_cnv1;
        MoveL Target_280,v1500,z100,ROBOBEL926_T_TD_300\WObj:=wobj_cnv1;
        MoveL Target_290,v1500,z100,ROBOBEL926_T_TD_300\WObj:=wobj_cnv1;
        MoveL Target_300,v1500,z100,ROBOBEL926_T_TD_300\WObj:=wobj_cnv1;
        MoveL Target_310,v1500,z100,ROBOBEL926_T_TD_300\WObj:=wobj_cnv1;
        MoveL Target_320,v1500,z100,ROBOBEL926_T_TD_300\WObj:=wobj_cnv1;
        MoveL Target_330,v1500,z100,ROBOBEL926_T_TD_300\WObj:=wobj_cnv1;
        MoveL Target_340,v1500,z100,ROBOBEL926_T_TD_300\WObj:=wobj_cnv1;
        MoveL Target_350,v1500,z100,ROBOBEL926_T_TD_300\WObj:=wobj_cnv1;
        MoveL Target_360,v1500,z100,ROBOBEL926_T_TD_300\WObj:=wobj_cnv1;
        MoveL Target_370,v1500,z100,ROBOBEL926_T_TD_300\WObj:=wobj_cnv1;
    ENDPROC
    PROC Path_30()
    ENDPROC
    PROC HOME()
        MoveL Target_410,v1000,z100,ROBOBEL926_T_TD_150\WObj:=wobj0;
    ENDPROC
    PROC Path_40()
        !HOME;
        MoveJ Target_390,v1000,z100,ROBOBEL926_T_TD_150\WObj:=Workobject_x;
        MoveJ Target_410,v1000,z100,ROBOBEL926_T_TD_150\WObj:=Workobject_x;
    ENDPROC
    PROC Paint_Lam()
    ENDPROC
    PROC Path_50()
        MoveJ Target_430,v1000,z100,ROBOBEL926_T_TD_150\WObj:=Workobject_x;
        MoveJ Target_410,v1000,z100,ROBOBEL926_T_TD_150\WObj:=Workobject_x;
    ENDPROC
    PROC Path_60()
        MoveJ Target_440,v1000,z100,ROBOBEL926_T_TD_150\WObj:=Workobject_x;
        MoveJ Target_510,v1000,z100,ROBOBEL926_T_TD_150\WObj:=Workobject_x;
        MoveJ Target_500,v1000,z100,ROBOBEL926_T_TD_150\WObj:=Workobject_x;
        MoveJ Target_410,v1000,z100,ROBOBEL926_T_TD_150\WObj:=Workobject_x;
    ENDPROC
ENDMODULE

--- Backups/Controlador_Pintura_v2/RAPID/TASK1/SYSMOD/cnvdata.sys ---
module cnvdata(sysmodule)

   pers wobjdata wobjtrack := [false,false,"CNV1",[[0,0,0],[1,0,0,0]],[[0,0,0],[1,0,0,0]]];



   proc DropWobjTrack()
      if OpMode() = OP_AUTO then
         if GetSignal("c1Connected") = 1 then
            DropWObj wobjtrack;
         endif
      endif
   endproc



   !-----------------------------------------------
   ! Synchronised Wait Work Object
   !
   ! This instruction does the following:
   !   1) Move to WaitPos relative to Wobj
   !   2) Keep robot in WaitPoint relative to Wobj until Wobj has
   !      reached RelDist
   !
   proc SyncWWObj(
      num RelDist,
      robtarget WaitPoint,
      inout tooldata Tool,
      inout wobjdata Wobj)

      var robtarget pWait;

      pWait := Offs(WaitPoint, 2, 0, 0);
      PaintL WaitPoint, v1000, z50, Tool \Wobj := Wobj;
      while (GetSignal("c1Position") * 1000) < RelDist do
        PaintL pWait, v5, z50, Tool \Wobj := Wobj;
        PaintL WaitPoint, v5, z50, Tool \Wobj := Wobj;
      endwhile
      PaintL pWait, v5, z50, Tool \Wobj := Wobj;
      return;
   backward
      PaintL WaitPoint, v300, z50, Tool \Wobj := Wobj;
   endproc



endmodule

--- Backups/Controlador_Pintura_v2/RAPID/TASK1/SYSMOD/ctsync.sys ---
module ctsync(sysmodule,nostepin)
   !
   ! (C) Copyright 2008 ABB
   !




   pers num nConvRamping := 0.2; ! User-configurable conveyor ramping characteristic.
   pers bool bCTSyncInfo := true;
   local const num MAX_STOP_TIME := 9;

   local var clock clkConv;
   var num nStopTime;
   local var intnum irConvStop;
   local var intnum irConvStart;
   local var intnum irReposFinished;
   local var signaldo doReposFinAlias;
   local var signaldo doNullSpeedAlias;
   local var signaldi diNullSpeedAlias;

   pers tooldata tCurrTool := [true,[[0,0,0],[1,0,0,0]],[0,[0,0,0],[1,0,0,0],0,0,0]];
   pers wobjdata wobjCurrWobj := [false,true,"",[[0,0,0],[1,0,0,0]],[[0,0,0],[1,0,0,0]]];



   proc InitCTSync()
      var string stReposFinished := "";

      ! Handle if c1NullSpeed is either a DI or a DO.
      InitNullSpeedDI;
      InitNullSpeedDO;

      if GetSignal("ReposFinished") <> -1000000 then
         stReposFinished := "ReposFinished";
         AliasIO stReposFinished, doReposFinAlias;

         IDelete irReposFinished;
         connect irReposFinished with tpReposFinished;
         ISignalDO doReposFinAlias, 1, irReposFinished;
      endif
   endproc



   proc InitNullSpeedDI()
      var string stNullSpeed := "";

      if GetSignal("c1NullSpeed") <> -1000000 then
         stNullSpeed := "c1NullSpeed";
         AliasIO stNullSpeed, diNullSpeedAlias;

         IDelete irConvStop;
         connect irConvStop with tpConvStop;
         ISignalDI diNullSpeedAlias, 1, irConvStop;

         IDelete irConvStart;
         connect irConvStart with tpConvStart;
         ISignalDI diNullSpeedAlias, 0, irConvStart;
      endif
   error
      if errno = ERR_ALIASIO_TYPE then
         SkipWarn;
         return;
      endif
   endproc



   proc InitNullSpeedDO()
      var string stNullSpeed := "";

      if GetSignal("c1NullSpeed") <> -1000000 then
         stNullSpeed := "c1NullSpeed";
         AliasIO stNullSpeed, doNullSpeedAlias;

         IDelete irConvStop;
         connect irConvStop with tpConvStop;
         ISignalDO doNullSpeedAlias, 1, irConvStop;

         IDelete irConvStart;
         connect irConvStart with tpConvStart;
         ISignalDO doNullSpeedAlias, 0, irConvStart;
      endif
   error
      if errno = ERR_ALIASIO_TYPE then
         SkipWarn;
         return;
      endif
   endproc



   proc ResetConvTime()
      nStopTime := 0;
      ClkStop clkConv;
      ClkReset clkConv;

      ! Make sure synchronization is off before starting a program.
      CnvSync \Off;
   endproc



   proc SyncPos(robtarget WaitPoint, num nCurrBrush \num RetractDist \num RelDist \Switch DirectionX | Switch DirectionY)
      var num nTempRetract;

      ! Only run in auto mode.
      ! Always retracts in manual mode, this is not preferred by the users.
      if OpMode() <> OP_AUTO
         return;

      if Present(RetractDist) then
         nTempRetract := RetractDist;
      else
         nTempRetract := 0;
      endif

      ! Can be called directly, or use wrapper instruction instead.
      if Present(RelDist) then
         if RelDist > c1Position * 1000 then
            if Present(DirectionX) then
               WaitConv WaitPoint, nCurrBrush, nTempRetract \RelDist := RelDist \DirectionX;
            elseif Present(DirectionY) then
               WaitConv WaitPoint, nCurrBrush, nTempRetract \RelDist := RelDist \DirectionY;
            else ! DirectionZ
               WaitConv WaitPoint, nCurrBrush, nTempRetract \RelDist := RelDist;
            endif
         endif
      else
         if nStopTime > MAX_STOP_TIME then
            nStopTime := MAX_STOP_TIME;
            if bCTSyncInfo
               ErrWrite \I, "Stop time too big (" + ValToStr(nStopTime) + "s)!", "Limited to " + ValToStr(MAX_STOP_TIME) + "s.";
         endif
         if c1NullSpeed = 1 or nStopTime > 3 then
            if Present(DirectionX) then
               WaitConv WaitPoint, nCurrBrush, nTempRetract \DirectionX;
            elseif Present(DirectionY) then
               WaitConv WaitPoint, nCurrBrush, nTempRetract \DirectionY;
            else ! DirectionZ
               WaitConv WaitPoint, nCurrBrush, nTempRetract;
            endif
         endif
      endif
   endproc



   local proc WaitConv(robtarget WaitPoint, num CurrBrush, num RetractDist \num RelDist \Switch DirectionX | Switch DirectionY)
      var robtarget pStopPaint;
      var robtarget pStopPaintOffset;
      var pos pTrigVect;
      var num nTrigAxis;
      var num nTrigValue;
      var num nRelDist;
      var num nLocalCnvPos;
      var num nConvSpeed;

      tCurrTool := CTool();
      wobjCurrWobj := CWObj();

      if Present(DirectionX) then
         pStopPaint := RelTool(WaitPoint, RetractDist, 0, 0);
      elseif Present(DirectionY) then
         pStopPaint := RelTool(WaitPoint, 0, RetractDist, 0);
      else ! DirectionZ
         ! Only allow retract in negative direction, for backwards compability.
         pStopPaint := RelTool(WaitPoint, 0, 0, 0 - Abs(RetractDist));
      endif

      pTrigVect := pStopPaint.trans - WaitPoint.trans;
      if Abs(pTrigVect.x) > Abs(pTrigVect.y) and Abs(pTrigVect.x) > Abs(pTrigVect.z) then
         nTrigAxis := 0;
         nTrigValue := WaitPoint.trans.x + pTrigVect.x / 4;
      elseif Abs(pTrigVect.y) > Abs(pTrigVect.z) then
         nTrigAxis := 1;
         nTrigValue := WaitPoint.trans.y + pTrigVect.y / 4;
      else
         nTrigAxis := 2;
         nTrigValue := WaitPoint.trans.z + pTrigVect.z / 4;
      endif

      ! WaitBrush is a system wide constant.
      if RetractDist <> 0 then
         if nTrigAxis = 0 then
            SetBrush WaitBrush \X := nTrigValue;
         elseif nTrigAxis = 1 then
            SetBrush WaitBrush \Y := nTrigValue;
         else
            SetBrush WaitBrush \Z := nTrigValue;
         endif
         PaintLSig pStopPaint, v500, fine, tCurrTool \Wobj := wobjCurrWobj;
      else
         PaintLSig WaitPoint, v500, fine, tCurrTool \Wobj := wobjCurrWobj; ! Prevent prefetch RAPID execution of SetBrush.
         SetBrush WaitBrush;
      endif

      ClkStop clkConv;
      if c1NullSpeed = 1
         nStopTime := nStopTime + ClkRead(clkConv) - 0.3;
      if nStopTime < 0.1
         nStopTime := 0.1;

      nLocalCnvPos := c1Position;

      if Present(RelDist) then
         nRelDist := RelDist;
      else
         nConvSpeed := PntCnvAvgSpeed();
         nRelDist := (nLocalCnvPos + (nStopTime * nConvSpeed)) * 1000;
      endif

      if bCTSyncInfo
         ErrWrite \I, "Wait Conveyor", "nRDist: " + ValToStr(nRelDist) + " c1Pos: " +  ValToStr(nLocalCnvPos) + " nStpTm: " + ValToStr(nStopTime) + " CnvSpd: " + ValToStr(nConvSpeed);

      ! WaitWObj wobjCurrWobj \RelDist := nRelDist;
      pStopPaintOffset := RelTool(pStopPaint, 0, 0, 0 - 2);
      while GetSignal("c1Position") < nRelDist / 1000 do
         if GetSignal("A1Brush") <> WaitBrush
            SetBrush WaitBrush; ! Prevent problem with Repos setting last brush after wait reached.
         PaintLSig pStopPaint, v500, z0, tCurrTool \Wobj := wobjCurrWobj;
         PaintLSig pStopPaintOffset, v500, z0, tCurrTool \Wobj := wobjCurrWobj;
      endwhile

      nStopTime := 0;
      ClkReset clkConv;

      if RetractDist <> 0 then
         if nTrigAxis = 0 then
            SetBrush CurrBrush \X := nTrigValue;
         elseif nTrigAxis = 1 then
            SetBrush CurrBrush \Y := nTrigValue;
         else
            SetBrush CurrBrush \Z := nTrigValue;
         endif
         PaintLSig WaitPoint, v500, z10, tCurrTool \Wobj := wobjCurrWobj;
      else
         PaintLSig WaitPoint, v500, fine, tCurrTool \Wobj := wobjCurrWobj;
         SetBrush CurrBrush;
      endif
   error
      trynext;
   endproc



   trap tpConvStop
      if GetSignal("doInModule") = 1 and GetSignal("doHomePos") = 0 and GetSignal("sdoCycleOn") = 1 then
         if bCTSyncInfo
            ErrWrite \I, "Conveyor Stopped", "Conveyor Stopped";
         ClkReset clkConv;
         ClkStart clkConv;
      endif
   endtrap



   trap tpConvStart
      if GetSignal("doInModule") = 1 and GetSignal("doHomePos") = 0 then
         ClkStop clkConv;
         nStopTime := nStopTime + ClkRead(clkConv) + nConvRamping;
         ClkReset clkConv;
         if bCTSyncInfo
            ErrWrite \I , "Conveyor Started", "StopTime: " + ValToStr(nStopTime);
      endif
   endtrap



   proc RobStop()
      if GetSignal("doInModule") = 1 and GetSignal("doHomePos") = 0 then
         ClkStop clkConv;
         nStopTime := nStopTime + ClkRead(clkConv) - 0.3;
         ClkReset clkConv;
      endif
   endproc



   proc RobStart()
      if OpMode() <> OP_AUTO
         return;
      if GetSignal("doInModule") = 1 and GetSignal("doHomePos") = 0 then
         ClkReset clkConv;
         ClkStart clkConv;
      endif
      if PPMovedInManMode() then
         nStopTime := 0;
         if bCTSyncInfo
            ErrWrite \I,  "PPMovedInManMode: RobStart", "StopTime: 0";
         ResetPPMoved;
      endif
   endproc



   trap tpReposFinished
      if GetSignal("doInModule") = 1 and GetSignal("doHomePos") = 0 then
         ClkReset clkConv;
         ClkStart clkConv;
         if bCTSyncInfo
            ErrWrite \I, "Repos Finished", "StopTime: " + ValToStr(nStopTime);
      endif
   endtrap



endmodule

--- Backups/Controlador_Pintura_v2/RAPID/TASK1/SYSMOD/custmain.sys ---
module custmain(sysmodule)



   proc InitCustMain()
      !
      ! Insert RAPID code for start at main here...
      !
   endproc



   proc PreMainCustom()
      !
      ! This will be executed before a paint program...
      !
   endproc



   proc PostMainCustom()
      !
      ! This will be executed after a paint program...
      !
   endproc



endmodule

--- Backups/Controlador_Pintura_v2/RAPID/TASK1/SYSMOD/robdata.sys ---
module robdata(sysmodule)

   ! Note: This file can be used to add custom tools and speeds.
   ! Uncomment any standard tools here, if they are needed.



   ! Default generic gun (10x5cm, 60 degree):
   pers tooldata tDefGun_Tip := [true,[[50,0,100],[0.866025,0,0.5,0]],[2,[0,0,50],[1,0,0,0],0,0,0]];
   pers tooldata tDefGun_100 := [true,[[136.6,0,150],[0.866025,0,0.5,0]],[2,[0,0,50],[1,0,0,0],0,0,0]];
   pers tooldata tDefGun_200 := [true,[[223.2,0,200],[0.866025,0,0.5,0]],[2,[0,0,50],[1,0,0,0],0,0,0]];

   ! Robobel 925:
   !pers tooldata tRB925_200 := [true,[[290.1,0,540],[0.866025,0,0.5,0]],[8,[0,0,33],[1,0,0,0],0,0,0]];
   !pers tooldata tRB925_250 := [true,[[333.4,0,565],[0.866025,0,0.5,0]],[8,[0,0,33],[1,0,0,0],0,0,0]];

   ! HCEBELL:
   !pers tooldata tHCEBELL_0   := [true,[[142.9,0,427.5],[0.866025,0,0.5,0]],[10,[0,-40,250],[1,0,0,0],0,0,0]];
   !pers tooldata tHCEBELL_150 := [true,[[272.8,0,502.5],[0.866025,0,0.5,0]],[11,[0,40,250],[1,0,0,0],0,0,0]];
   !pers tooldata tHCEBELL_200 := [true,[[316.1,0,527.5],[0.866025,0,0.5,0]],[11,[0,40,250],[1,0,0,0],0,0,0]];
   !pers tooldata tHCEBELL_250 := [true,[[359.4,0,552.5],[0.866025,0,0.5,0]],[11,[0,40,250],[1,0,0,0],0,0,0]];
   !pers tooldata tHCEBELL_300 := [true,[[402.7,0,577.5],[0.866025,0,0.5,0]],[11,[0,40,250],[1,0,0,0],0,0,0]];

   ! ABB Ecco Gun:
   !pers tooldata tEccoGun_Tip := [true,[[1.8,0,156.6],[0.965926,0,0.258819,0]],[2,[0,0,120],[1,0,0,0],0,0,0]];
   !pers tooldata tEccoGun_200 := [true,[[101.8,0,329.8],[0.965926,0,0.258819,0]],[2,[0,0,120],[1,0,0,0],0,0,0]];
   !pers tooldata tEccoGun_250 := [true,[[126.8,0,373.1],[0.965926,0,0.258819,0]],[2,[0,0,120],[1,0,0,0],0,0,0]];
   !pers tooldata tEccoGun_300 := [true,[[151.8,0,416.4],[0.965926,0,0.258819,0]],[2,[0,0,120],[1,0,0,0],0,0,0]];

   ! G1Direct (short bracket):
   !pers tooldata tG1Direct_300 := [true,[[571.58,0,450],[0.866025,0,0.5,0]],[6.6,[135.2,0,174.1],[1,0,0,0],0,0,0]];
   !pers tooldata tG1Direct_250 := [true,[[528.28,0,425],[0.866025,0,0.5,0]],[6.6,[135.2,0,174.1],[1,0,0,0],0,0,0]];
   !pers tooldata tG1Direct_200 := [true,[[484.97,0,400],[0.866025,0,0.5,0]],[6.6,[135.2,0,174.1],[1,0,0,0],0,0,0]];

   ! G1_Long Braket:
   !pers tooldata tG1V3_200L := [true,[[487,0,502.3],[0.866025,0,0.5,0]],[8,[140.6,0,170],[1,0,0,0],0,0,0]];
   !pers tooldata tG1V3_250L := [true,[[524,0,528.9],[0.866025,0,0.5,0]],[8,[140.6,0,170],[1,0,0,0],0,0,0]];
   !pers tooldata tG1V3_300L := [true,[[549,0,571.6],[0.866025,0,0.5,0]],[8,[140.6,0,170],[1,0,0,0],0,0,0]];

   ! Cartridge Bell:
   !pers tooldata tCBS_0   := [true,[[121.25,0,415],[0.866025,0,0.5,0]],[5.5,[30,0,225],[1,0,0,0],0,0,0]];
   !pers tooldata tCBS_100 := [true,[[207.85,0,465],[0.866025,0,0.5,0]],[5.5,[30,0,225],[1,0,0,0],0,0,0]];
   !pers tooldata tCBS_200 := [true,[[294.45,0,515],[0.866025,0,0.5,0]],[5.5,[30,0,225],[1,0,0,0],0,0,0]];
   !pers tooldata tCBS_250 := [true,[[337.75,0,540],[0.866025,0,0.5,0]],[5.5,[30,0,225],[1,0,0,0],0,0,0]];
   !pers tooldata tCBS_300 := [true,[[381.05,0,565],[0.866025,0,0.5,0]],[5.5,[30,0,225],[1,0,0,0],0,0,0]];

   ! Cartridge Gun:
   !pers tooldata tCGS_0   := [true,[[127.44,0,418.5],[0.866025,0,0.5,0]],[8.1,[30,0,225],[1,0,0,0],0,0,0]];
   !pers tooldata tCGS_100 := [true,[[214.04,0,468.5],[0.866025,0,0.5,0]],[8.1,[30,0,225],[1,0,0,0],0,0,0]];
   !pers tooldata tCGS_200 := [true,[[300.64,0,518.5],[0.866025,0,0.5,0]],[8.1,[30,0,225],[1,0,0,0],0,0,0]];
   !pers tooldata tCGS_250 := [true,[[343.95,0,543.5],[0.866025,0,0.5,0]],[8.1,[30,0,225],[1,0,0,0],0,0,0]];
   !pers tooldata tCGS_300 := [true,[[387.11,0,568.5],[0.866025,0,0.5,0]],[8.1,[30,0,225],[1,0,0,0],0,0,0]];

   ! Robobel 926:
   !pers tooldata tRB926TD_0   := [true,[[116.9,0,470],[0.866025,0,0.5,0]],[5.5,[30,0,225],[1,0,0,0],0,0,0]];
   !pers tooldata tRB926TD_100 := [true,[[203.5,0,520],[0.866025,0,0.5,0]],[5.5,[30,0,225],[1,0,0,0],0,0,0]];
   !pers tooldata tRB926TD_120 := [true,[[220.8,0,530],[0.866025,0,0.5,0]],[5.5,[30,0,225],[1,0,0,0],0,0,0]];
   !pers tooldata tRB926TD_150 := [true,[[246.8,0,545],[0.866025,0,0.5,0]],[5.5,[30,0,225],[1,0,0,0],0,0,0]];
   !pers tooldata tRB926TD_200 := [true,[[290.1,0,570],[0.866025,0,0.5,0]],[5.5,[30,0,225],[1,0,0,0],0,0,0]];
   !pers tooldata tRB926TD_250 := [true,[[333.4,0,595],[0.866025,0,0.5,0]],[5.5,[30,0,225],[1,0,0,0],0,0,0]];
   !pers tooldata tRB926TD_300 := [true,[[376.7,0,620],[0.866025,0,0.5,0]],[5.5,[30,0,225],[1,0,0,0],0,0,0]];

   ! Robobel 625TD:
   !pers tooldata tRB625TD_0   := [true,[[116.9,0,420],[0.866025,0,0.5,0]],[5.1,[30,0,215],[1,0,0,0],0,0,0]];
   !pers tooldata tRB625TD_150 := [true,[[246.8,0,495],[0.866025,0,0.5,0]],[5.1,[30,0,215],[1,0,0,0],0,0,0]];
   !pers tooldata tRB625TD_200 := [true,[[290.1,0,520],[0.866025,0,0.5,0]],[5.1,[30,0,215],[1,0,0,0],0,0,0]];
   !pers tooldata tRB625TD_250 := [true,[[333.4,0,545],[0.866025,0,0.5,0]],[5.1,[30,0,215],[1,0,0,0],0,0,0]];
   !pers tooldata tRB625TD_300 := [true,[[376.7,0,570],[0.866025,0,0.5,0]],[5.1,[30,0,215],[1,0,0,0],0,0,0]];

   ! Robobel 951TD:
   !pers tooldata tRB951TD_0   := [true,[[116.9,0,470],[0.866025,0,0.5,0]],[6.3,[30,0,220],[1,0,0,0],0,0,0]];
   !pers tooldata tRB951TD_100 := [true,[[203.5,0,520],[0.866025,0,0.5,0]],[6.3,[30,0,220],[1,0,0,0],0,0,0]];
   !pers tooldata tRB951TD_120 := [true,[[220.8,0,530],[0.866025,0,0.5,0]],[6.3,[30,0,220],[1,0,0,0],0,0,0]];
   !pers tooldata tRB951TD_150 := [true,[[246.8,0,545],[0.866025,0,0.5,0]],[6.3,[30,0,220],[1,0,0,0],0,0,0]];
   !pers tooldata tRB951TD_200 := [true,[[290.1,0,570],[0.866025,0,0.5,0]],[6.3,[30,0,220],[1,0,0,0],0,0,0]];
   !pers tooldata tRB951TD_250 := [true,[[333.4,0,595],[0.866025,0,0.5,0]],[6.3,[30,0,220],[1,0,0,0],0,0,0]];
   !pers tooldata tRB951TD_300 := [true,[[376.7,0,620],[0.866025,0,0.5,0]],[6.3,[30,0,220],[1,0,0,0],0,0,0]];

   ! Robobel 951CBS /40pai/50pai/70pai:
   !pers tooldata tRB951CBS_0   := [true,[[121.25,0,415],[0.866025,0,0.5,0]],[6.3,[55,0,225],[1,0,0,0],0,0,0]];
   !pers tooldata tRB951CBS_100 := [true,[[207.85,0,465],[0.866025,0,0.5,0]],[6.3,[55,0,225],[1,0,0,0],0,0,0]];
   !pers tooldata tRB951CBS_120 := [true,[[225.17,0,475],[0.866025,0,0.5,0]],[6.3,[55,0,225],[1,0,0,0],0,0,0]];
   !pers tooldata tRB951CBS_150 := [true,[[251.15,0,490],[0.866025,0,0.5,0]],[6.3,[55,0,225],[1,0,0,0],0,0,0]];
   !pers tooldata tRB951CBS_200 := [true,[[294.45,0,515],[0.866025,0,0.5,0]],[6.3,[55,0,225],[1,0,0,0],0,0,0]];
   !pers tooldata tRB951CBS_250 := [true,[[337.75,0,540],[0.866025,0,0.5,0]],[6.3,[55,0,225],[1,0,0,0],0,0,0]];
   !pers tooldata tRB951CBS_300 := [true,[[381.05,0,565],[0.866025,0,0.5,0]],[6.3,[55,0,225],[1,0,0,0],0,0,0]];

   ! Interior Robobel951CBS /30pai:
   !pers tooldata tInteriorCBS_0   := [true,[[99.6,0,402.5],[0.866025,0,0.5,0]],[6.3,[30,0,220],[1,0,0,0],0,0,0]];
   !pers tooldata tInteriorCBS_100 := [true,[[186.2,0,452.5],[0.866025,0,0.5,0]],[6.3,[30,0,220],[1,0,0,0],0,0,0]];
   !pers tooldata tInteriorCBS_120 := [true,[[246.8,0,487.5],[0.866025,0,0.5,0]],[6.3,[30,0,220],[1,0,0,0],0,0,0]];
   !pers tooldata tInteriorCBS_150 := [true,[[272.8,0,502.5],[0.866025,0,0.5,0]],[6.3,[30,0,220],[1,0,0,0],0,0,0]];
   !pers tooldata tInteriorCBS_200 := [true,[[316.1,0,527.5],[0.866025,0,0.5,0]],[6.3,[30,0,220],[1,0,0,0],0,0,0]];
   !pers tooldata tInteriorCBS_250 := [true,[[359.4,0,552.5],[0.866025,0,0.5,0]],[6.3,[30,0,220],[1,0,0,0],0,0,0]];
   !pers tooldata tInteriorCBS_300 := [true,[[402.7,0,577.5],[0.866025,0,0.5,0]],[6.3,[30,0,220],[1,0,0,0],0,0,0]];

   ! Interior Robobel951 /30pai:
   !pers tooldata tInterior951_0   := [true,[[138.6,0,482.5],[0.866025,0,0.5,0]],[6.3,[30,0,220],[1,0,0,0],0,0,0]];
   !pers tooldata tInterior951_100 := [true,[[225.17,0,532.5],[0.866025,0,0.5,0]],[6.3,[30,0,220],[1,0,0,0],0,0,0]];
   !pers tooldata tInterior951_120 := [true,[[242.49,0,542.5],[0.866025,0,0.5,0]],[6.3,[30,0,220],[1,0,0,0],0,0,0]];
   !pers tooldata tInterior951_150 := [true,[[268.47,0,557.5],[0.866025,0,0.5,0]],[6.3,[30,0,220],[1,0,0,0],0,0,0]];
   !pers tooldata tInterior951_200 := [true,[[311.77,0,582.5],[0.866025,0,0.5,0]],[6.3,[30,0,220],[1,0,0,0],0,0,0]];
   !pers tooldata tInterior951_250 := [true,[[355.07,0,607.5],[0.866025,0,0.5,0]],[6.3,[30,0,220],[1,0,0,0],0,0,0]];
   !pers tooldata tInterior951_300 := [true,[[398.37,0,632.5],[0.866025,0,0.5,0]],[6.3,[30,0,220],[1,0,0,0],0,0,0]];

   ! RB-1000WSC (700cc Cartridge):
   !pers tooldata tRB1000WSC_0     := [true,[[121.25,0,450],[0.866025,0,0.5,0]],[13.0,[-52,0,270],[1,0,0,0],0,0,0]];
   !pers tooldata tRB1000WSC_100   := [true,[[207.85,0,500],[0.866025,0,0.5,0]],[13.0,[-52,0,270],[1,0,0,0],0,0,0]];
   !pers tooldata tRB1000WSC_150   := [true,[[251.15,0,525],[0.866025,0,0.5,0]],[13.0,[-52,0,270],[1,0,0,0],0,0,0]];
   !pers tooldata tRB1000WSC_200   := [true,[[294.45,0,550],[0.866025,0,0.5,0]],[13.0,[-52,0,270],[1,0,0,0],0,0,0]];
   !pers tooldata tRB1000WSC_250   := [true,[[337.75,0,575],[0.866025,0,0.5,0]],[13.0,[-52,0,270],[1,0,0,0],0,0,0]];
   !pers tooldata tRB1000WSC_300   := [true,[[381.05,0,600],[0.866025,0,0.5,0]],[13.0,[-52,0,270],[1,0,0,0],0,0,0]];
   !pers tooldata tRB1000WSC_teach := [true,[[-259.801,0,230],[0.866025,0,0.5,0]],[13.0,[-52,0,270],[1,0,0,0],0,0,0]];

   ! RB-1000SAD (Robobel Type):
   !pers tooldata tRB1000SAD_0   := [true,[[181.9,0,472.5],[0.866025,0,0.5,0]],[10.7,[31,0,260],[1,0,0,0],0,0,0]];
   !pers tooldata tRB1000SAD_100 := [true,[[268.5,0,522.5],[0.866025,0,0.5,0]],[10.7,[31,0,260],[1,0,0,0],0,0,0]];
   !pers tooldata tRB1000SAD_150 := [true,[[311.8,0,547.5],[0.866025,0,0.5,0]],[10.7,[31,0,260],[1,0,0,0],0,0,0]];
   !pers tooldata tRB1000SAD_200 := [true,[[355.1,0,572.5],[0.866025,0,0.5,0]],[10.7,[31,0,260],[1,0,0,0],0,0,0]];
   !pers tooldata tRB1000SAD_250 := [true,[[398.4,0,597.5],[0.866025,0,0.5,0]],[10.7,[31,0,260],[1,0,0,0],0,0,0]];
   !pers tooldata tRB1000SAD_300 := [true,[[441.7,0,622.5],[0.866025,0,0.5,0]],[10.7,[31,0,260],[1,0,0,0],0,0,0]];

   ! RB-1000SSD (Robobel Type):
   !pers tooldata tRB1000SSD_0   := [true,[[181.9,0,472.5],[0.866025,0,0.5,0]],[10.7,[31,0,260],[1,0,0,0],0,0,0]];
   !pers tooldata tRB1000SSD_100 := [true,[[268.5,0,522.5],[0.866025,0,0.5,0]],[10.7,[31,0,260],[1,0,0,0],0,0,0]];
   !pers tooldata tRB1000SSD_150 := [true,[[311.8,0,547.5],[0.866025,0,0.5,0]],[10.7,[31,0,260],[1,0,0,0],0,0,0]];
   !pers tooldata tRB1000SSD_200 := [true,[[355.1,0,572.5],[0.866025,0,0.5,0]],[10.7,[31,0,260],[1,0,0,0],0,0,0]];
   !pers tooldata tRB1000SSD_250 := [true,[[398.4,0,597.5],[0.866025,0,0.5,0]],[10.7,[31,0,260],[1,0,0,0],0,0,0]];
   !pers tooldata tRB1000SSD_300 := [true,[[441.7,0,622.5],[0.866025,0,0.5,0]],[10.7,[31,0,260],[1,0,0,0],0,0,0]];

   ! RoboBel021-mini for HollowWrist
   !pers tooldata tRB1021min_tip := [true,[[170.0,0,200],[0.866025,0,0.5,0]],[2.8,[80,0,140],[1,0,0,0],0,0,0]];
   !pers tooldata tRB1021min_100 := [true,[[256.6,0,250],[0.866025,0,0.5,0]],[2.8,[80,0,140],[1,0,0,0],0,0,0]];
   !pers tooldata tRB1021min_150 := [true,[[299.9,0,275],[0.866025,0,0.5,0]],[2.8,[80,0,140],[1,0,0,0],0,0,0]];
   !pers tooldata tRB1021min_200 := [true,[[343.2,0,300],[0.866025,0,0.5,0]],[2.8,[80,0,140],[1,0,0,0],0,0,0]];
   !pers tooldata tRB1021min_250 := [true,[[386.5,0,325],[0.866025,0,0.5,0]],[2.8,[80,0,140],[1,0,0,0],0,0,0]];
   !pers tooldata tRB1021min_300 := [true,[[429.8,0,350],[0.866025,0,0.5,0]],[2.8,[80,0,140],[1,0,0,0],0,0,0]];
   !pers tooldata tRB1021min_350 := [true,[[473.1,0,375],[0.866025,0,0.5,0]],[2.8,[80,0,140],[1,0,0,0],0,0,0]];
   !pers tooldata tRB1021min_400 := [true,[[516.4,0,400],[0.866025,0,0.5,0]],[2.8,[80,0,140],[1,0,0,0],0,0,0]];

   ! AGMD PRO gun with single attachment for Hollow wrist. No Dump (3HNM 10123-1)
   !pers tooldata tAGP10123_TIP:=[TRUE,[[ 52,0,198],[0.866025,0,0.5,0]],[1.490,[0, 0, 101],[1,0,0,0],0,0,0]];
   !pers tooldata tAGP10123_150:=[TRUE,[[178,0,273],[0.866025,0,0.5,0]],[1.490,[0, 0, 101],[1,0,0,0],0,0,0]];
   !pers tooldata tAGP10123_225:=[TRUE,[[243,0,310],[0.866025,0,0.5,0]],[1.490,[0, 0, 101],[1,0,0,0],0,0,0]];
   !pers tooldata tAGP10123_300:=[TRUE,[[308,0,348],[0.866025,0,0.5,0]],[1.490,[0, 0, 101],[1,0,0,0],0,0,0]];

   ! AGMD PRO gun with single attachment for Hollow wrist. With Dump. (3HNM 10121-1)
   !pers tooldata tAGP10121_TIP:=[TRUE,[[ 52,0,198],[0.866025,0,0.5,0]],[1.510,[0, 0, 100],[1,0,0,0],0,0,0]];
   !pers tooldata tAGP10121_150:=[TRUE,[[178,0,273],[0.866025,0,0.5,0]],[1.510,[0, 0, 100],[1,0,0,0],0,0,0]];
   !pers tooldata tAGP10121_225:=[TRUE,[[243,0,310],[0.866025,0,0.5,0]],[1.510,[0, 0, 100],[1,0,0,0],0,0,0]];
   !pers tooldata tAGP10121_300:=[TRUE,[[308,0,348],[0.866025,0,0.5,0]],[1.510,[0, 0, 100],[1,0,0,0],0,0,0]];

   ! AGMD PRO gun with single attachment for Hollow wirst. With Dump, MPAC version. (3HNA 017776-001)
   !pers tooldata tAGP17776_TIP:=[TRUE,[[ 52,0,198],[0.866025,0,0.5,0]],[1.520,[0,0,103],[1,0,0,0],0,0,0]];
   !pers tooldata tAGP17776_150:=[TRUE,[[178,0,273],[0.866025,0,0.5,0]],[1.520,[0,0,103],[1,0,0,0],0,0,0]];
   !pers tooldata tAGP17776_225:=[TRUE,[[243,0,310],[0.866025,0,0.5,0]],[1.520,[0,0,103],[1,0,0,0],0,0,0]];
   !pers tooldata tAGP17776_300:=[TRUE,[[308,0,348],[0.866025,0,0.5,0]],[1.520,[0,0,103],[1,0,0,0],0,0,0]];

   ! RB1000-EXT Short Bracket
   !pers tooldata tRB1000EXTS_TIP:=[TRUE,[[362.5,0,121.0],[0.866025,0,0.5,0]],[10.2,[130, 0, 182],[1,0,0,0],0,0,0]];
   !pers tooldata tRB1000EXTS_100:=[TRUE,[[400.5,0,352.2],[0.866025,0,0.5,0]],[10.2,[130, 0, 182],[1,0,0,0],0,0,0]];
   !pers tooldata tRB1000EXTS_200:=[TRUE,[[487.1,0,402.2],[0.866025,0,0.5,0]],[10.2,[130, 0, 182],[1,0,0,0],0,0,0]];
   !pers tooldata tRB1000EXTS_250:=[TRUE,[[530.4,0,427.2],[0.866025,0,0.5,0]],[10.2,[130, 0, 182],[1,0,0,0],0,0,0]];
   !pers tooldata tRB1000EXTS_300:=[TRUE,[[573.7,0,452.2],[0.866025,0,0.5,0]],[10.2,[130, 0, 182],[1,0,0,0],0,0,0]];

   ! RB1000-EXT Long Bracket
   !pers tooldata tRB1000EXTL_TIP:=[TRUE,[[362.5,0,221.0],[0.866025,0,0.5,0]],[10.6,[130, 0, 260],[1,0,0,0],0,0,0]];
   !pers tooldata tRB1000EXTL_100:=[TRUE,[[400.5,0,452.2],[0.866025,0,0.5,0]],[10.6,[130, 0, 260],[1,0,0,0],0,0,0]];
   !pers tooldata tRB1000EXTL_200:=[TRUE,[[487.1,0,502.2],[0.866025,0,0.5,0]],[10.6,[130, 0, 260],[1,0,0,0],0,0,0]];
   !pers tooldata tRB1000EXTL_250:=[TRUE,[[530.4,0,527.2],[0.866025,0,0.5,0]],[10.6,[130, 0, 260],[1,0,0,0],0,0,0]];
   !pers tooldata tRB1000EXTL_300:=[TRUE,[[573.7,0,552.2],[0.866025,0,0.5,0]],[10.6,[130, 0, 260],[1,0,0,0],0,0,0]];

   ! RB1000i-SSD
   !pers tooldata tRB1000iSSD_TIP:=[TRUE,[[228.6,0,480.0],[0.866025,0,0.5,0]],[9.0,[52, 0, 293],[1,0,0,0],0,0,0]];
   !pers tooldata tRB1000iSSD_100:=[TRUE,[[315.2,0,530.0],[0.866025,0,0.5,0]],[9.0,[52, 0, 293],[1,0,0,0],0,0,0]];
   !pers tooldata tRB1000iSSD_200:=[TRUE,[[401.8,0,580.0],[0.866025,0,0.5,0]],[9.0,[52, 0, 293],[1,0,0,0],0,0,0]];
   !pers tooldata tRB1000iSSD_250:=[TRUE,[[445.1,0,605.0],[0.866025,0,0.5,0]],[9.0,[52, 0, 293],[1,0,0,0],0,0,0]];
   !pers tooldata tRB1000iSSD_300:=[TRUE,[[488.4,0,630.0],[0.866025,0,0.5,0]],[9.0,[52, 0, 293],[1,0,0,0],0,0,0]];

   ! RB1000i-SAD
   !pers tooldata tRB1000iSAD_TIP:=[TRUE,[[228.6,0,480.0],[0.866025,0,0.5,0]],[9.0,[52, 0, 293],[1,0,0,0],0,0,0]];
   !pers tooldata tRB1000iSAD_100:=[TRUE,[[315.2,0,530.0],[0.866025,0,0.5,0]],[9.0,[52, 0, 293],[1,0,0,0],0,0,0]];
   !pers tooldata tRB1000iSAD_200:=[TRUE,[[401.8,0,580.0],[0.866025,0,0.5,0]],[9.0,[52, 0, 293],[1,0,0,0],0,0,0]];
   !pers tooldata tRB1000iSAD_250:=[TRUE,[[445.1,0,605.0],[0.866025,0,0.5,0]],[9.0,[52, 0, 293],[1,0,0,0],0,0,0]];
   !pers tooldata tRB1000iSAD_300:=[TRUE,[[488.4,0,630.0],[0.866025,0,0.5,0]],[9.0,[52, 0, 293],[1,0,0,0],0,0,0]];

   ! RB1000i-S2K
   !pers tooldata tRB1000iS2K_TIP:=[TRUE,[[228.6,0,480.0],[0.866025,0,0.5,0]],[9.0,[52, 0, 293],[1,0,0,0],0,0,0]];
   !pers tooldata tRB1000iS2K_100:=[TRUE,[[315.2,0,530.0],[0.866025,0,0.5,0]],[9.0,[52, 0, 293],[1,0,0,0],0,0,0]];
   !pers tooldata tRB1000iS2K_200:=[TRUE,[[401.8,0,580.0],[0.866025,0,0.5,0]],[9.0,[52, 0, 293],[1,0,0,0],0,0,0]];
   !pers tooldata tRB1000iS2K_250:=[TRUE,[[445.1,0,605.0],[0.866025,0,0.5,0]],[9.0,[52, 0, 293],[1,0,0,0],0,0,0]];
   !pers tooldata tRB1000iS2K_300:=[TRUE,[[488.4,0,630.0],[0.866025,0,0.5,0]],[9.0,[52, 0, 293],[1,0,0,0],0,0,0]];

   ! RB1000i External charge, Long Bracket
   !pers tooldata tRB1000iEXTL_TIP:=[TRUE,[[313.9,0,402.3],[0.866025,0,0.5,0]],[11.3,[128.5, 0, 266],[1,0,0,0],0,0,0]];
   !pers tooldata tRB1000iEXTL_100:=[TRUE,[[400.5,0,452.3],[0.866025,0,0.5,0]],[11.3,[128.5, 0, 266],[1,0,0,0],0,0,0]];
   !pers tooldata tRB1000iEXTL_200:=[TRUE,[[487.1,0,502.3],[0.866025,0,0.5,0]],[11.3,[128.5, 0, 266],[1,0,0,0],0,0,0]];
   !pers tooldata tRB1000iEXTL_250:=[TRUE,[[530.4,0,527.3],[0.866025,0,0.5,0]],[11.3,[128.5, 0, 266],[1,0,0,0],0,0,0]];
   !pers tooldata tRB1000iEXTL_300:=[TRUE,[[573.7,0,552.3],[0.866025,0,0.5,0]],[11.3,[128.5, 0, 266],[1,0,0,0],0,0,0]];

   ! RB1000i External charge, Short Bracket
   !pers tooldata tRB1000iEXTS_TIP:=[TRUE,[[313.9,0,302.3],[0.866025,0,0.5,0]],[10.8,[136.6, 0, 188.4],[1,0,0,0],0,0,0]];
   !pers tooldata tRB1000iEXTS_100:=[TRUE,[[400.5,0,352.3],[0.866025,0,0.5,0]],[10.8,[136.6, 0, 188.4],[1,0,0,0],0,0,0]];
   !pers tooldata tRB1000iEXTS_200:=[TRUE,[[487.1,0,402.3],[0.866025,0,0.5,0]],[10.8,[136.6, 0, 188.4],[1,0,0,0],0,0,0]];
   !pers tooldata tRB1000iEXTS_250:=[TRUE,[[530.4,0,427.3],[0.866025,0,0.5,0]],[10.8,[136.6, 0, 188.4],[1,0,0,0],0,0,0]];
   !pers tooldata tRB1000iEXTS_300:=[TRUE,[[573.7,0,452.3],[0.866025,0,0.5,0]],[10.8,[136.6, 0, 188.4],[1,0,0,0],0,0,0]];

   ! RB1000-CE (Compact External)
   !pers tooldata tRB1000CE_TIP:=[TRUE,[[233.8,0,370.0],[0.866025,0,0.5,0]],[9.5,[72, 0, 236],[1,0,0,0],0,0,0]];
   !pers tooldata tRB1000CE_100:=[TRUE,[[320.4,0,420.0],[0.866025,0,0.5,0]],[9.5,[72, 0, 236],[1,0,0,0],0,0,0]];
   !pers tooldata tRB1000CE_200:=[TRUE,[[407.0,0,470.0],[0.866025,0,0.5,0]],[9.5,[72, 0, 236],[1,0,0,0],0,0,0]];
   !pers tooldata tRB1000CE_250:=[TRUE,[[450.3,0,495.0],[0.866025,0,0.5,0]],[9.5,[72, 0, 236],[1,0,0,0],0,0,0]];
   !pers tooldata tRB1000CE_300:=[TRUE,[[493.6,0,520.0],[0.866025,0,0.5,0]],[9.5,[72, 0, 236],[1,0,0,0],0,0,0]];

   ! RB1000i-WSC 300cc cartridge.
   !pers tooldata tRB1000iWSC300_tip:=[TRUE,[[160.2,0,501.5],[0.866025,0,0.5,0]],[13.2,[-40.32, 0,290],[1,0,0,0],0,0,0]];
   !pers tooldata tRB1000iWSC300_100:=[TRUE,[[246.8,0,551.5],[0.866025,0,0.5,0]],[13.2,[-40.32, 0,290],[1,0,0,0],0,0,0]];
   !pers tooldata tRB1000iWSC300_200:=[TRUE,[[333.4,0,601.5],[0.866025,0,0.5,0]],[13.2,[-40.32, 0,290],[1,0,0,0],0,0,0]];
   !pers tooldata tRB1000iWSC300_300:=[TRUE,[[420.0,0,651.5],[0.866025,0,0.5,0]],[13.2,[-40.32, 0,290],[1,0,0,0],0,0,0]];

   ! RB1000i-WSC 500cc cartridge.
   !pers tooldata tRB1000iWSC500_tip:=[TRUE,[[160.2,0,501.5],[0.866025,0,0.5,0]],[13.7,[-30.17, 0,292.1],[1,0,0,0],0,0,0]];
   !pers tooldata tRB1000iWSC500_100:=[TRUE,[[246.8,0,551.5],[0.866025,0,0.5,0]],[13.7,[-30.17, 0,292.1],[1,0,0,0],0,0,0]];
   !pers tooldata tRB1000iWSC500_200:=[TRUE,[[333.4,0,601.5],[0.866025,0,0.5,0]],[13.7,[-30.17, 0,292.1],[1,0,0,0],0,0,0]];
   !pers tooldata tRB1000iWSC500_300:=[TRUE,[[420.0,0,651.5],[0.866025,0,0.5,0]],[13.7,[-30.17, 0,292.1],[1,0,0,0],0,0,0]];

   ! RB1000i-WSC 700cc cartridge.
   !pers tooldata tRB1000iWSC700_tip:=[TRUE,[[160.2,0,501.5],[0.866025,0,0.5,0]],[14.2,[-21.46, 0,293.46],[1,0,0,0],0,0,0]];
   !pers tooldata tRB1000iWSC700_100:=[TRUE,[[246.8,0,551.5],[0.866025,0,0.5,0]],[14.2,[-21.46, 0,293.46],[1,0,0,0],0,0,0]];
   !pers tooldata tRB1000iWSC700_200:=[TRUE,[[333.4,0,601.5],[0.866025,0,0.5,0]],[14.2,[-21.46, 0,293.46],[1,0,0,0],0,0,0]];
   !pers tooldata tRB1000iWSC700_300:=[TRUE,[[420.0,0,651.5],[0.866025,0,0.5,0]],[14.2,[-21.46, 0,293.46],[1,0,0,0],0,0,0]];

   ! RB1000i-CE (Short Bracket)
   !pers tooldata tRB1000iCE_TIP := [true,[[233.80,0,305],[0.866025,0,0.5,0]],[9.6,[69.5,0,183.1],[1,0,0,0],0,0,0]];
   !pers tooldata tRB1000iCE_100 := [true,[[320.40,0,355],[0.866025,0,0.5,0]],[9.6,[69.5,0,183.1],[1,0,0,0],0,0,0]];
   !pers tooldata tRB1000iCE_200 := [true,[[407.01,0,405],[0.866025,0,0.5,0]],[9.6,[69.5,0,183.1],[1,0,0,0],0,0,0]];
   !pers tooldata tRB1000iCE_250 := [true,[[450.30,0,430],[0.866025,0,0.5,0]],[9.6,[69.5,0,183.1],[1,0,0,0],0,0,0]];
   !pers tooldata tRB1000iCE_300 := [true,[[493.60,0,455],[0.866025,0,0.5,0]],[9.6,[69.5,0,183.1],[1,0,0,0],0,0,0]];

   ! RB1000i-CE (Long Bracket)
   !pers tooldata tRB1000iCEL_TIP := [true,[[233.80,0,370],[0.866025,0,0.5,0]],[10,[67.8,0,233],[1,0,0,0],0,0,0]];
   !pers tooldata tRB1000iCEL_100 := [true,[[320.40,0,420],[0.866025,0,0.5,0]],[10,[67.8,0,233],[1,0,0,0],0,0,0]];
   !pers tooldata tRB1000iCEL_150 := [true,[[363.70,0,445],[0.866025,0,0.5,0]],[10,[67.8,0,233],[1,0,0,0],0,0,0]];
   !pers tooldata tRB1000iCEL_200 := [true,[[407.01,0,470],[0.866025,0,0.5,0]],[10,[67.8,0,233],[1,0,0,0],0,0,0]];
   !pers tooldata tRB1000iCEL_250 := [true,[[450.30,0,495],[0.866025,0,0.5,0]],[10,[67.8,0,233],[1,0,0,0],0,0,0]];
   !pers tooldata tRB1000iCEL_300 := [true,[[493.60,0,520],[0.866025,0,0.5,0]],[10,[67.8,0,233],[1,0,0,0],0,0,0]];

   ! RoboBel031 on IRB580 bracket.
   !pers tooldata tRB031PC580_tip := [true,[[170.0,0,300.0],[0.866025,0,0.5,0]],[3.3,[72.8,0,200],[1,0,0,0],0,0,0]];
   !pers tooldata tRB031PC580_100 := [true,[[256.6,0,350.0],[0.866025,0,0.5,0]],[3.3,[72.8,0,200],[1,0,0,0],0,0,0]];
   !pers tooldata tRB031PC580_200 := [true,[[343.2,0,400.0],[0.866025,0,0.5,0]],[3.3,[72.8,0,200],[1,0,0,0],0,0,0]];
   !pers tooldata tRB031PC580_300 := [true,[[429.8,0,450.0],[0.866025,0,0.5,0]],[3.3,[72.8,0,200],[1,0,0,0],0,0,0]];

   ! PixelPaint inkjet print head.
   !pers tooldata tPrintHead_tip := [true,[[304.49,0,336.4],[0.866025,0,0.5,0]],[13,[150,0,168],[1,0,0,0],0,0,0]];
   !pers tooldata tPrintHead_005 := [true,[[308.82,0,338.9],[0.866025,0,0.5,0]],[13,[150,0,168],[1,0,0,0],0,0,0]];
   !pers tooldata tPrintHead_010 := [true,[[313.36,0,341.5],[0.866025,0,0.5,0]],[13,[150,0,168],[1,0,0,0],0,0,0]];

   ! RB1000i-S SSD/SAD/S2K.
   !pers tooldata tRB1000iS_tip := [true,[[236.4,0,484.5],[0.866025,0,0.5,0]],[8.8,[50,0,293.5],[1,0,0,0],0,0,0]];
   !pers tooldata tRB1000iS_100 := [true,[[323.0,0,534.5],[0.866025,0,0.5,0]],[8.8,[50,0,293.5],[1,0,0,0],0,0,0]];
   !pers tooldata tRB1000iS_110 := [true,[[331.7,0,539.5],[0.866025,0,0.5,0]],[8.8,[50,0,293.5],[1,0,0,0],0,0,0]];
   !pers tooldata tRB1000iS_120 := [true,[[340.3,0,544.5],[0.866025,0,0.5,0]],[8.8,[50,0,293.5],[1,0,0,0],0,0,0]];
   !pers tooldata tRB1000iS_130 := [true,[[349.0,0,549.5],[0.866025,0,0.5,0]],[8.8,[50,0,293.5],[1,0,0,0],0,0,0]];
   !pers tooldata tRB1000iS_140 := [true,[[357.7,0,554.5],[0.866025,0,0.5,0]],[8.8,[50,0,293.5],[1,0,0,0],0,0,0]];
   !pers tooldata tRB1000iS_150 := [true,[[366.3,0,559.5],[0.866025,0,0.5,0]],[8.8,[50,0,293.5],[1,0,0,0],0,0,0]];
   !pers tooldata tRB1000iS_200 := [true,[[409.6,0,584.5],[0.866025,0,0.5,0]],[8.8,[50,0,293.5],[1,0,0,0],0,0,0]];



   ! Speed data:
   !const speeddata vPaint50   := [50,300,1000,50];
   !const speeddata vPaint100  := [100,300,100,100];
   !const speeddata vPaint150  := [150,300,150,150];
   !const speeddata vPaint200  := [200,300,200,200];
   !const speeddata vPaint250  := [250,300,250,250];
   !const speeddata vPaint300  := [300,300,300,300];
   !const speeddata vPaint350  := [350,300,350,350];
   !const speeddata vPaint400  := [400,300,400,400];
   !const speeddata vPaint450  := [450,300,450,450];
   !const speeddata vPaint500  := [500,300,500,500];
   !const speeddata vPaint550  := [550,300,1000,500];
   !const speeddata vPaint600  := [600,300,1000,500];
   !const speeddata vPaint650  := [650,300,1000,500];
   !const speeddata vPaint700  := [700,300,1000,500];
   !const speeddata vPaint750  := [750,300,1000,500];
   !const speeddata vPaint800  := [800,300,1000,500];
   !const speeddata vPaint850  := [850,300,1000,500];
   !const speeddata vPaint900  := [900,300,1000,500];
   !const speeddata vPaint950  := [950,300,1000,500];
   !const speeddata vPaint1000 := [1000,300,1000,500];
   !const speeddata vPaint1100 := [1100,300,1000,500];
   !const speeddata vPaint1200 := [1200,300,1000,500];
   !const speeddata vPaint1300 := [1300,300,1000,500];
   !const speeddata vPaint1400 := [1400,300,1000,500];
   !const speeddata vPaint1500 := [1500,300,1000,500];
   !const speeddata vPaint1600 := [1600,300,1000,500];
   !const speeddata vPaint1700 := [1700,300,1000,500];
   !const speeddata vPaint1800 := [1800,300,1000,500];
   !const speeddata vPaint1900 := [1900,300,1000,500];
   !const speeddata vPaint2000 := [2000,300,1000,500];
   !const speeddata vPaint2100 := [2100,300,1000,500];
   !const speeddata vPaint2200 := [2200,300,1000,500];
   !const speeddata vPaint2300 := [2300,300,1000,500];
   !const speeddata vPaint2400 := [2400,300,1000,500];
   !const speeddata vPaint2500 := [2500,300,1000,500];



   ! Speed data (High Flow Bell):
   const speeddata vHFB50   := [50,150,50,50];
   const speeddata vHFB100  := [100,150,100,100];
   const speeddata vHFB150  := [150,150,150,150];
   const speeddata vHFB200  := [200,150,200,200];
   const speeddata vHFB250  := [250,150,250,250];
   const speeddata vHFB300  := [300,150,300,300];
   const speeddata vHFB350  := [350,150,350,350];
   const speeddata vHFB400  := [400,150,400,400];
   const speeddata vHFB450  := [450,150,450,450];
   const speeddata vHFB500  := [500,150,500,500];
   const speeddata vHFB550  := [550,150,1000,500];
   const speeddata vHFB600  := [600,150,1000,500];
   const speeddata vHFB650  := [650,150,1000,500];
   const speeddata vHFB700  := [700,150,1000,500];
   const speeddata vHFB750  := [750,150,1000,500];
   const speeddata vHFB800  := [800,150,1000,500];
   const speeddata vHFB850  := [850,150,1000,500];
   const speeddata vHFB900  := [900,150,1000,500];
   const speeddata vHFB950  := [950,150,1000,500];
   const speeddata vHFB1000 := [1000,150,1000,500];
   const speeddata vHFB1100 := [1100,150,1000,500];
   const speeddata vHFB1200 := [1200,150,1000,500];
   const speeddata vHFB1300 := [1300,150,1000,500];
   const speeddata vHFB1400 := [1400,150,1000,500];
   const speeddata vHFB1500 := [1500,150,1000,500];
   const speeddata vHFB1600 := [1600,150,1000,500];
   const speeddata vHFB1700 := [1700,150,1000,500];
   const speeddata vHFB1800 := [1800,150,1000,500];
   const speeddata vHFB1900 := [1900,150,1000,500];
   const speeddata vHFB2000 := [2000,150,1000,500];
   const speeddata vHFB2100 := [2100,150,1000,500];
   const speeddata vHFB2200 := [2200,150,1000,500];
   const speeddata vHFB2300 := [2300,150,1000,500];
   const speeddata vHFB2400 := [2400,150,1000,500];
   const speeddata vHFB2500 := [2500,150,1000,500];



   ! Zone data:
   !const zonedata zPaint1   := [false,1,1,1,0.15,1,0.15];
   !const zonedata zPaint5   := [false,5,8,8,0.8,8,0.8];
   !const zonedata zPaint10  := [false,10,15,15,1.5,15,1.5];
   !const zonedata zPaint15  := [false,15,23,23,2.3,23,2.3];
   !const zonedata zPaint20  := [false,20,30,30,3,30,3];
   !const zonedata zPaint30  := [false,30,45,45,4.5,45,4.5];
   !const zonedata zPaint40  := [false,40,60,60,6,60,6];
   !const zonedata zPaint50  := [false,50,75,75,7.5,75,7.5];
   !const zonedata zPaint60  := [false,60,90,90,9,90,9];
   !const zonedata zPaint80  := [false,80,120,120,12,120,12];
   !const zonedata zPaint100 := [false,100,150,150,15,150,15];
   !const zonedata zPaint150 := [false,150,225,225,23,225,23];
   !const zonedata zPaint200 := [false,200,300,300,30,300,30];
   !const zonedata zPaint250 := [false,250,375,375,37.5,375,37.5];
   !const zonedata zPaint300 := [false,300,450,450,45,450,45];



endmodule

--- Backups/Controlador_Pintura_v2/RAPID/TASK1/SYSMOD/sysdata.sys ---
module sysdata(sysmodule)

   ! Note: This file is used to store system positions and setup world zones.



   pers tooldata tUserTool0 := [TRUE,[[0,0,0],[1,0,0,0]],[0.001,[0,0,0.001],[1,0,0,0],0,0,0]];

   pers robtarget pHomePos   := [[0,0,0],[9E+09,9E+09,9E+09,9E+09],[-1,-1,1,0],[9E+09,9E+09,9E+09,9E+09,9E+09,9E+09]];
   pers robtarget pMtrlChPos := [[0,0,0],[9E+09,9E+09,9E+09,9E+09],[-1,-1,1,0],[9E+09,9E+09,9E+09,9E+09,9E+09,9E+09]];
   pers robtarget pReadyPos  := [[0,0,0],[9E+09,9E+09,9E+09,9E+09],[-1,-1,1,0],[9E+09,9E+09,9E+09,9E+09,9E+09,9E+09]];
   pers robtarget pUserPos   := [[0,0,0],[9E+09,9E+09,9E+09,9E+09],[-1,-1,1,0],[9E+09,9E+09,9E+09,9E+09,9E+09,9E+09]];

   pers jointtarget jHomePos   := [[9E+09,9E+09,9E+09,9E+09,9E+09,9E+09],[9E+09,9E+09,9E+09,9E+09,9E+09,0]];
   pers jointtarget jMtrlChPos := [[9E+09,9E+09,9E+09,9E+09,9E+09,9E+09],[9E+09,9E+09,9E+09,9E+09,9E+09,0]];
   pers jointtarget jReadyPos  := [[9E+09,9E+09,9E+09,9E+09,9E+09,9E+09],[9E+09,9E+09,9E+09,9E+09,9E+09,0]];
   pers jointtarget jUserPos   := [[9E+09,9E+09,9E+09,9E+09,9E+09,9E+09],[9E+09,9E+09,9E+09,9E+09,9E+09,0]];

   local var wzstationary wzHomePos;
   local var wzstationary wzMtrlChPos;
   local var wzstationary wzReadyPos;
   local var wzstationary wzUserPos;

   local var pos psHomePos   := [0,0,0];
   local var pos psMtrlChPos := [0,0,0];
   local var pos psReadyPos  := [0,0,0];
   local var pos psUserPos   := [0,0,0];

   local var signaldo doHomePosAlias;
   local var signaldo doMtrlChPosAlias;
   local var signaldo doReadyPosAlias;
   local var signaldo doUserPosAlias;



   proc PowerOnWZones()
      var shapedata volHomePos;
      var shapedata volMtrlChPos;
      var shapedata volReadyPos;
      var shapedata volUserPos;

      ! AliasIO requires variables to work.
      var string stHomePos       := "doHomePos";
      var string stMtrlChangePos := "doMtrlChangePos";
      var string stReadyPos      := "doReadyPos";
      var string stUserPos       := "doUserPos";

      psHomePos   := pHomePos.trans;
      psMtrlChPos := pMtrlChPos.trans;
      psReadyPos  := pReadyPos.trans;
      psUserPos   := pUserPos.trans;

      WZSphDef \Inside, volHomePos, psHomePos, 6;
      WZSphDef \Inside, volMtrlChPos, psMtrlChPos, 6;
      WZSphDef \Inside, volReadyPos, psReadyPos, 6;
      WZSphDef \Inside, volUserPos, psUserPos, 6;

      if GetSignal("doHomePos") <> -1000000 then
         AliasIO stHomePos, doHomePosAlias;
         WZDOSet \Stat, wzHomePos \Inside, volHomePos, doHomePosAlias, 1;
      endif
      if GetSignal("doMtrlChangePos") <> -1000000 then
         AliasIO stMtrlChangePos, doMtrlChPosAlias;
         WZDOSet \Stat, wzMtrlChPos \Inside, volMtrlChPos, doMtrlChPosAlias, 1;
      endif
      if GetSignal("doReadyPos") <> -1000000 then
         AliasIO stReadyPos, doReadyPosAlias;
         WZDOSet \Stat, wzReadyPos \Inside, volReadyPos, doReadyPosAlias, 1;
      endif
      if GetSignal("doUserPos") <> -1000000 then
         AliasIO stUserPos, doUserPosAlias;
         WZDOSet \Stat, wzUserPos \Inside, volUserPos, doUserPosAlias, 1;
      endif
   endproc



   proc ConfSettingsOff()
      ConfJ \Off;
      ConfL \Off;
   endproc



endmodule

--- Backups/Controlador_Pintura_v2/RAPID/TASK2/SYSMOD/custcmd.sys ---
module custcmd(sysmodule)



   proc InitCustCmd()
      !
      ! Insert RAPID code for startup here...
      !
   endproc



   proc Cmd1001(num nInParam{*}, inout num nResult, inout num nOutData{*})
      !
      ! Insert RAPID code for command here...
      !
      ErrWrite "Cmd1001",
         ValToStr(nInParam{1}) + "," +
         ValToStr(nInParam{2}) + "," +
         ValToStr(nInParam{3}) + "," +
         ValToStr(nInParam{4}) + "," +
         ValToStr(nInParam{5}) + "," +
         ValToStr(nInParam{6}) + "," +
         ValToStr(nInParam{7}) + "," +
         ValToStr(nInParam{8}) + "," +
         ValToStr(nInParam{9}) + "," +
         ValToStr(nInParam{10});

      nResult := CMD_OK;
   endproc



   proc Cmd1002(num nInParam{*}, inout num nResult, inout num nOutData{*})
      !
      ! Insert RAPID code for command here...
      !
      ErrWrite "Cmd1002", "";

      nOutData{1}  := nInParam{1};
      nOutData{2}  := nInParam{2};
      nOutData{3}  := nInParam{3};
      nOutData{4}  := nInParam{4};
      nOutData{5}  := nInParam{5};
      nOutData{6}  := nInParam{6};
      nOutData{7}  := nInParam{7};
      nOutData{8}  := nInParam{8};
      nOutData{9}  := nInParam{9};
      nOutData{10} := nInParam{10};

      nResult := CMD_OK;
   endproc



endmodule

--- Backups/Controlador_Pintura_v2/HOME/programs/calpos.mod ---
module calpos

   ! SCOPE: Universal calibration/sync position program.

   proc mainCalPos()
      var jointtarget jLocalCalPos;

      ! Dummy instruction for SetPP.
      WaitTime 1;

      ! Set default values for all axis.
      jLocalCalPos := [[9E+09,9E+09,9E+09,9E+09,9E+09,9E+09],[9E+09,9E+09,9E+09,9E+09,9E+09,0]];

      jLocalCalPos.robax.rax_1 := nArmCalPos("rob1_1");
      jLocalCalPos.robax.rax_2 := nArmCalPos("rob1_2");
      jLocalCalPos.robax.rax_3 := nArmCalPos("rob1_3");
      jLocalCalPos.robax.rax_4 := nArmCalPos("rob1_4");
      jLocalCalPos.robax.rax_5 := nArmCalPos("rob1_5");
      jLocalCalPos.robax.rax_6 := nArmCalPos("rob1_6");

      if nRobSerialPart() = 5500 or nRobSerialPart() = 5510 then
         ! IRB5500 and IRB5510 has special values on axis 5 and 6, just set to 0 as stated in the manual.
         jLocalCalPos.robax.rax_5 := 0;
         jLocalCalPos.robax.rax_6 := 0;
      endif

      if stSingleJoint("AX7_1") <> "" then
         ! 7-axis robot.
         jLocalCalPos.extax.eax_a := nArmCalPos(stSingleJoint("AX7_1") \NoConversion)*1000;
      elseif nArmCalPos("obp_3") <> 9E+09 then
         ! 3-axis TurnTable.
         !IndReset OBP,2\RefNum:=0\Short;
         !IndReset OBP,3\RefNum:=0\Short;
         jLocalCalPos.extax.eax_a := nArmCalPos("obp_1");
         jLocalCalPos.extax.eax_b := nArmCalPos("obp_2");
         jLocalCalPos.extax.eax_c := nArmCalPos("obp_3");
      elseif nArmCalPos("obp_2") <> 9E+09 then
         ! 2-axis TurnTable.
         jLocalCalPos.extax.eax_a := nArmCalPos("obp_1");
         jLocalCalPos.extax.eax_b := nArmCalPos("obp_2");
      elseif nArmCalPos("obp_1") <> 9E+09 then
         ! 1-axis TurnTable.
         jLocalCalPos.extax.eax_a := nArmCalPos("obp_1");
      elseif nArmCalPos("track1") <> 9E+09 then
         ! IRB5350-02.
         jLocalCalPos.robax.rax_4 := 0;
         jLocalCalPos.robax.rax_5 := 0;
         jLocalCalPos.robax.rax_6 := 0;
         jLocalCalPos.extax.eax_a := nArmCalPos("track1" \NoConversion);
      elseif stRobotType() = "ROB1_5350_01_T00F82_A21C21D21" then
         ! IRB5350-01.
         jLocalCalPos.robax.rax_4 := 0;
         jLocalCalPos.robax.rax_5 := 0;
         jLocalCalPos.robax.rax_6 := 0;
      elseif stRobotAx7Type() = "PNT_5500_ROT_AX7" then
         ! IRB5500-27.
         jLocalCalPos.extax.eax_a := 0;
         jLocalCalPos.extax.eax_b := 0;
      else
         ! Attempt to get values for 8-axis robot.
         jLocalCalPos.extax.eax_a := nArmCalPos("rob1_7" \NoConversion);
         jLocalCalPos.extax.eax_b := nArmCalPos("rob1_8" \NoConversion);
      endif

      if stSingleJoint("H1AngleAxis") <> "" then
         ! Global CBS.
         jLocalCalPos.extax.eax_b := 0;
         jLocalCalPos.extax.eax_c := 0;
         jLocalCalPos.extax.eax_d := 0;
         jLocalCalPos.extax.eax_e := 0;
      endif

      MoveAbsJ jLocalCalPos,v100,fine,tool0;
      Stop;
   endproc

   local func num nArmCalPos(string stArm \switch NoConversion)
      var num nCalPos;
      ReadCfgData "/MOC/ARM/" + stArm, "cal_position", nCalPos;
      if Present(NoConversion) then
         return nCalPos;
      else
         return Round(nCalPos * (180 / 3.1415926) \Dec := 3);
      endif
   error
      if errno = ERR_CFG_NOTFND then
         SkipWarn;
         return 9E+09;
      endif
   endfunc

   local func string stSingleJoint(string stSingle)
      var string stJoint;
      ReadCfgData "/MOC/SINGLE/" + stSingle, "use_joint", stJoint;
      return stJoint;
   error
      if errno = ERR_CFG_NOTFND then
         SkipWarn;
         return "";
      endif
   endfunc

   local func num nRobSerialPart()
      var string stPart;
      var num nPart;
      ReadCfgData "/MOC/ROBOT_SERIAL_NUMBER/PID", "robot_serial_number_high_part", stPart;
      if StrToVal(StrPart(stPart, 1, StrFind(stPart, 1, "_") - 1), nPart) then
         return nPart;
      else
         return 9E+09;
      endif
   error
      SkipWarn;
      return 9E+09;
   endfunc

   local func string stRobotType()
      var string stType;
      ReadCfgData "/MOC/ROBOT/ROB_1", "use_robot_type", stType;
      return stType;
   error
      if errno = ERR_CFG_NOTFND then
         SkipWarn;
         return "";
      endif
   endfunc

   local func string stRobotAx7Type()
      var string stType;
      ReadCfgData "/MOC/ROBOT/ROT_AX7", "use_robot_type", stType;
      return stType;
   error
      if errno = ERR_CFG_NOTFND then
         SkipWarn;
         return "";
      endif
   endfunc

endmodule

--- Backups/Controlador_Pintura_v2/HOME/programs/m1.mod ---
MODULE M1

  PROC mainM1()
    WaitTime 10;
  ENDPROC

ENDMODULE

--- Backups/Controlador_Pintura_v2/HOME/programs/m10001.mod ---
module m10001

   ! SCOPE: Motion program for home position.

   proc mainm10001()
      if jHomePos.robax.rax_1 = 9E+09 then
         ErrWrite \W, "Home position not taught!", "";
      else
         MoveAbsJ jHomePos,v300,fine,tUserTool0;
      endif
   endproc

endmodule

--- Backups/Controlador_Pintura_v2/HOME/programs/m2.mod ---
MODULE M2

  PROC mainM2()
    WaitTime 10;
  ENDPROC

ENDMODULE

--- Backups/Controlador_Pintura_v2/HOME/programs/m3.mod ---
MODULE M3

  PROC mainM3()
    WaitTime 10;
  ENDPROC

ENDMODULE

--- Backups/Controlador_Pintura_v2/SYSPAR/EIO.cfg ---
EIO:CFG_1.0:6:1::
#
SYSSIG_OUT:

      -Status "AutoOn" -Signal "AutoModeOn"

      -Status "RunchOk" -Signal "RunChainClosed"

      -Status "Error" -Signal "sdoRobotError"

      -Status "CycleOn" -Signal "sdoCycleOn"

      -Status "EmStop" -Signal "EmergencyStop"

      -Status "MotOnState" -Signal "MotorIsOn"

      -Status "WriteAccess" -Signal "MasterGranted"

      -Status "MotSupTrigg" -Signal "MotionSupTrigg"
#
SYSSIG_IN:

      -Signal "sdoAckAutoMode" -Action "AckAutoMode"

      -Signal "sdoResetError" -Action "ResetError"

      -Signal "sdoStartMain" -Action "StartMain"

      -Signal "sdoMotOnStart" -Action "MotOnStart"

      -Signal "sdoStop" -Action "Stop"

      -Signal "sdoQuickStop" -Action "QuickStop"

      -Signal "sdoMotorOn" -Action "MotorOn"

      -Signal "sdoMotorOff" -Action "MotorOff"

      -Signal "sdoWriteRequest" -Action "WriteAccess"
#
INDUSTRIAL_NETWORK:

      -Name "DeviceNet" -Label "DeviceNet Master/Slave Network" -Address "2"
#
EIO_CROSS:

      -Name "ReadyToReceiveCross" -Res "ReadyToReceive" -Act1 "doQueueFull"\
      -Act1_invert

      -Name "JobPendingCross" -Res "JobPending" -Act1 "doQueueEmpty"\
      -Act1_invert

      -Name "MtrlChRunningCross" -Res "MtrlChRunning" -Act1 "doMCSuspended"\
      -Act1_invert

      -Name "AppEnabledCross" -Res "AppEnabled" -Act1 "A1Enable"

      -Name "AppErrorCross" -Res "AppError" -Act1 "A1Error"

      -Name "HVEnabledCross" -Res "HVEnabled" -Act1 "A1HVEn" -Oper1 "AND"\
      -Act2 "READY_HV_ON"

      -Name "PotLifeWarningCross" -Res "PotLifeWarning" -Act1 "A1FluidPlWS"

      -Name "PotLifeTimeOutCross" -Res "PotLifeTimeOut" -Act1 "A1FluidPlTO"

      -Name "HomePosCross" -Res "HomePos" -Act1 "doHomePos"

      -Name "MtrlChangePosCross" -Res "MtrlChangePos" -Act1 "doMtrlChangePos"

      -Name "ReadyPosCross" -Res "ReadyPos" -Act1 "doReadyPos"

      -Name "UserPosCross" -Res "UserPos" -Act1 "doUserPos"

      -Name "doSwitchInAutoCross" -Res "doSwitchInAuto" -Act1 "AUTO1"\
      -Oper1 "AND" -Act2 "AUTO2"

      -Name "GoingToAutoCross" -Res "GoingToAuto" -Act1 "doSwitchInAuto"\
      -Oper1 "AND" -Act2 "AutoModeOn" -Act2_invert

      -Name "ReadyHighPriCross" -Res "ReadyHighPri" -Act1 "sdoCycleOn"\
      -Oper1 "AND" -Act2 "JobInProgress" -Act2_invert

      -Name "SystemRunningCross" -Res "SystemRunning" -Act1 "sdoCycleOn"\
      -Oper1 "AND" -Act2 "doQueuePause" -Act2_invert

      -Name "RobotErrorCross" -Res "RobotError" -Act1 "sdoRobotError"\
      -Oper1 "OR" -Act2 "doPntRapidError"

      -Name "BellRotatingCross" -Res "BellRotating" -Act1 "A1BellRotating"

      -Name "IPSNodesReadyCross" -Res "IPSNodesReady" -Act1 "NODES_UNREADY"\
      -Act1_invert

      -Name "ObjConnectedCross" -Res "ObjConnected" -Act1 "c1Connected"

      -Name "ConveyorRunningCross" -Res "ConveyorRunning" -Act1 "c1NullSpeed"\
      -Act1_invert
#
DEVICENET_DEVICE:

      -Name "Qtrack1" -Simulated  -VendorName "ABB Robotics"\
      -ProductName "Qtracker" -Address 15 -ProductCode 16 -DeviceType 100\
      -PollRate 20 -OutputSize 6 -InputSize 19
#
DEVICENET_COMMAND:

      -Name "CountsPerMeter1" -Device "Qtrack1" -OrderNr 2\
      -Path "6,20 66 24 01 30 01,CA,4" -Value "20000.0"

      -Name "SyncSeparation1" -Device "Qtrack1" -OrderNr 3\
      -Path "6,20 66 24 01 30 02,CA,4" -Value "0.005"

      -Name "QueueTrckDist1" -Device "Qtrack1" -OrderNr 4\
      -Path "6,20 66 24 01 30 03,CA,4" -Value "0.0"

      -Name "StartWinWidth1" -Device "Qtrack1" -OrderNr 5\
      -Path "6,20 66 24 01 30 04,CA,4" -Value "10.0"

      -Name "AutoBackup1" -Device "Qtrack1" -OrderNr 6\
      -Path "6,20 66 24 01 30 12,C1,1" -Value "1"

      -Name "SimulationVel1" -Device "Qtrack1" -OrderNr 7\
      -Path "6,20 66 24 01 30 13,CA,4" -Value "0.100"

      -Name "ScalingFactor1" -Device "Qtrack1" -OrderNr 8\
      -Path "6,20 66 24 01 30 14,CA,4" -Value "2000.0"

      -Name "CheckPointDist1" -Device "Qtrack1" -OrderNr 9\
      -Path "6,20 66 24 01 30 15,CA,4" -Value "0.0"

      -Name "CheckPWinWidth1" -Device "Qtrack1" -OrderNr 10\
      -Path "6,20 66 24 01 30 16,CA,4" -Value "0.0"

      -Name "IIRFPeriod1" -Device "Qtrack1" -OrderNr 11\
      -Path "6,20 66 24 01 30 05,CA,4" -Value "0.02"

      -Name "IIRFNoOfPoles1" -Device "Qtrack1" -OrderNr 12\
      -Path "6,20 66 24 01 30 06,C6,1" -Value "2"

      -Name "IIRFNoOfZeroes1" -Device "Qtrack1" -OrderNr 13\
      -Path "6,20 66 24 01 30 07,C6,1" -Value "0"

      -Name "IIRFXfrmMetPol1" -Device "Qtrack1" -OrderNr 14\
      -Path "6,20 66 24 01 30 08,C6,1" -Value "1"

      -Name "IIRFXfrmMetZero1" -Device "Qtrack1" -OrderNr 15\
      -Path "6,20 66 24 01 30 09,C6,1" -Value "1"

      -Name "IIRFFZ1" -Device "Qtrack1" -OrderNr 16\
      -Path "6,20 66 24 01 30 0A,CA,4" -Value "0.0"

      -Name "IIRFDZ1" -Device "Qtrack1" -OrderNr 17\
      -Path "6,20 66 24 01 30 0B,CA,4" -Value "0.0"

      -Name "IIRFFP1" -Device "Qtrack1" -OrderNr 18\
      -Path "6,20 66 24 01 30 0C,CA,4" -Value "2.0"

      -Name "IIRFDP1" -Device "Qtrack1" -OrderNr 19\
      -Path "6,20 66 24 01 30 0D,CA,4" -Value "0.707"

      -Name "IIRFGain1" -Device "Qtrack1" -OrderNr 20\
      -Path "6,20 66 24 01 30 0E,CA,4" -Value "1.0"

      -Name "FIRFLength1" -Device "Qtrack1" -OrderNr 21\
      -Path "6,20 66 24 01 30 0F,C6,1" -Value "0"

      -Name "FIRFB01" -Device "Qtrack1" -OrderNr 22\
      -Path "6,20 66 24 01 30 10,CA,4" -Value "0.0"

      -Name "FIRFB11" -Device "Qtrack1" -OrderNr 23\
      -Path "6,20 66 24 01 30 11,CA,4" -Value "0.0"
#
DEVICENET_INTERNAL_DEVICE:

      -Name "DN_Internal_Device" -VendorName "ABB Robotics"\
      -ProductName "DeviceNet Internal Slave Device"
#
ICI_DEVICE:

      -Name "PIB" -Network "ICI" -Label "Process Interface Board"\
      -Address "192.168.126.200"
#
EIO_SIGNAL:

      -Name "c1Position" -SignalType "AI" -Device "Qtrack1" -DeviceMap "0-31"\
      -MaxLog 21474.8 -MaxPhys 1 -MaxPhysLimit 1 -MaxBitVal 2147483647\
      -MinLog -21474.8 -MinPhys -1 -MinPhysLimit -1 -MinBitVal -2147483647

      -Name "c1Speed" -SignalType "AI" -Device "Qtrack1" -DeviceMap "32-63"\
      -MaxLog 21474.8 -MaxPhys 1 -MaxPhysLimit 1 -MaxBitVal 2147483647\
      -MinLog -21474.8 -MinPhys -1 -MinPhysLimit -1 -MinBitVal -2147483647

      -Name "c1Connected" -SignalType "DI" -Device "Qtrack1" -DeviceMap "104"

      -Name "c1NullSpeed" -SignalType "DI" -Device "Qtrack1" -DeviceMap "105"

      -Name "c1DReady" -SignalType "DI" -Device "Qtrack1" -DeviceMap "106"

      -Name "c1PassStw" -SignalType "DI" -Device "Qtrack1" -DeviceMap "107"

      -Name "c1NewObjStrobe" -SignalType "DI" -Device "Qtrack1" -DeviceMap "108"

      -Name "c1EncSelected" -SignalType "DI" -Device "Qtrack1" -DeviceMap "109"

      -Name "c1EncAFautlt" -SignalType "DI" -Device "Qtrack1" -DeviceMap "110"

      -Name "c1EncBFautlt" -SignalType "DI" -Device "Qtrack1" -DeviceMap "111"

      -Name "c1Simulating" -SignalType "DI" -Device "Qtrack1" -DeviceMap "112"

      -Name "c1DirOfTravel" -SignalType "DI" -Device "Qtrack1" -DeviceMap "113"

      -Name "c1ScaleEncPuls" -SignalType "DI" -Device "Qtrack1" -DeviceMap "114"

      -Name "c1PowerUpStatus" -SignalType "DI" -Device "Qtrack1" -DeviceMap "83"

      -Name "c1WaitWObj" -SignalType "DO" -Device "Qtrack1" -DeviceMap "0"

      -Name "c1DropWObj" -SignalType "DO" -Device "Qtrack1" -DeviceMap "1"

      -Name "c1Rem1PObj" -SignalType "DO" -Device "Qtrack1" -DeviceMap "2"

      -Name "c1RemAllPObj" -SignalType "DO" -Device "Qtrack1" -DeviceMap "3"

      -Name "c1EncSelect" -SignalType "DO" -Device "Qtrack1" -DeviceMap "4"

      -Name "c1SoftSyncSig" -SignalType "DO" -Device "Qtrack1" -DeviceMap "5"

      -Name "c1SoftCheckSig" -SignalType "DO" -Device "Qtrack1" -DeviceMap "6"

      -Name "c1SimMode" -SignalType "DO" -Device "Qtrack1" -DeviceMap "7"

      -Name "c1CntToEncStr" -SignalType "DO" -Device "Qtrack1" -DeviceMap "40"

      -Name "c1ForceJob" -SignalType "DO" -Device "Qtrack1" -DeviceMap "41"

      -Name "c1PosInJobQ" -SignalType "DO" -Device "Qtrack1" -DeviceMap "42"

      -Name "c1ObjectsInQ" -SignalType "GI" -Device "Qtrack1" -DeviceMap "64-71"

      -Name "c1CntFromEnc" -SignalType "GI" -Device "Qtrack1"\
      -DeviceMap "72-103"

      -Name "c1DTimestamp" -SignalType "GI" -Device "Qtrack1"\
      -DeviceMap "120-151"

      -Name "c1CntToEnc" -SignalType "GO" -Device "Qtrack1" -DeviceMap "8-39"

      -Name "AutoModeOn" -SignalType "DO"

      -Name "MasterGranted" -SignalType "DO"

      -Name "RunChainClosed" -SignalType "DO"

      -Name "RobotError" -SignalType "DO"

      -Name "JobInProgress" -SignalType "DO"

      -Name "JobPending" -SignalType "DO"

      -Name "ReadyHighPri" -SignalType "DO"

      -Name "SystemRunning" -SignalType "DO"

      -Name "MtrlChRunning" -SignalType "DO"

      -Name "MtrlChangeOn" -SignalType "DO"

      -Name "ObjConnected" -SignalType "DO"

      -Name "MtrlSupplyError" -SignalType "DO"

      -Name "AppEnabled" -SignalType "DO"

      -Name "AppError" -SignalType "DO"

      -Name "HVEnabled" -SignalType "DO"

      -Name "HVError" -SignalType "DO"

      -Name "PotLifeWarning" -SignalType "DO"

      -Name "PotLifeTimeOut" -SignalType "DO"

      -Name "HomePos" -SignalType "DO"

      -Name "MtrlChangePos" -SignalType "DO"

      -Name "ReadyPos" -SignalType "DO"

      -Name "UserPos" -SignalType "DO"

      -Name "ReposFinished" -SignalType "DO"

      -Name "EmergencyStop" -SignalType "DO"

      -Name "JobComplete" -SignalType "DO"

      -Name "GoingToAuto" -SignalType "DO"

      -Name "ReadyToReceive" -SignalType "DO"

      -Name "MotorIsOn" -SignalType "DO"

      -Name "ConveyorRunning" -SignalType "DO"

      -Name "ProgramLoaded" -SignalType "DO"

      -Name "CBSMotorIsOn" -SignalType "DO"

      -Name "BellRotating" -SignalType "DO"

      -Name "MotionSupTrigg" -SignalType "DO"

      -Name "PowerError" -SignalType "DO"

      -Name "IPSNodesReady" -SignalType "DO"

      -Name "doQueueFull" -SignalType "DO"

      -Name "doQueueEmpty" -SignalType "DO"

      -Name "doQueuePause" -SignalType "DO"

      -Name "doInModule" -SignalType "DO"

      -Name "doMCSuspended" -SignalType "DO"

      -Name "A1Enable" -SignalType "DO" -Access "All"

      -Name "A1Error" -SignalType "DO" -Access "All"

      -Name "A1HVEn" -SignalType "DO" -Access "All"

      -Name "A1FluidPlWS" -SignalType "DO" -Access "All"

      -Name "A1FluidPlTO" -SignalType "DO" -Access "All"

      -Name "doHomePos" -SignalType "DO" -Access "ReadOnly"

      -Name "doMtrlChangePos" -SignalType "DO" -Access "ReadOnly"

      -Name "doReadyPos" -SignalType "DO" -Access "ReadOnly"

      -Name "doUserPos" -SignalType "DO" -Access "ReadOnly"

      -Name "doSwitchInAuto" -SignalType "DO"

      -Name "doPntRapidError" -SignalType "DO"

      -Name "sdoRobotError" -SignalType "DO"

      -Name "sdoAckAutoMode" -SignalType "DO"

      -Name "sdoResetError" -SignalType "DO"

      -Name "sdoStartMain" -SignalType "DO"

      -Name "sdoMotOnStart" -SignalType "DO"

      -Name "sdoStop" -SignalType "DO"

      -Name "sdoQuickStop" -SignalType "DO"

      -Name "sdoMotorOn" -SignalType "DO"

      -Name "sdoMotorOff" -SignalType "DO"

      -Name "sdoCycleOn" -SignalType "DO"

      -Name "sdoWriteRequest" -SignalType "DO"

      -Name "A1Brush" -SignalType "GO" -Access "All"

      -Name "A1BrushTabNdx" -SignalType "GO" -Access "All"

      -Name "A1HVErrNo" -SignalType "GO" -Access "All"

      -Name "A1Material" -SignalType "GO" -Access "All"

      -Name "A1Fluid" -SignalType "AO" -Access "All"

      -Name "A1FluidAccu" -SignalType "AO" -Access "All"

      -Name "A1FluidEn" -SignalType "DO" -Access "All"

      -Name "A1NeedleEn" -SignalType "DO" -Access "All"

      -Name "A1BellRotating" -SignalType "DI" -Access "All"

      -Name "A1BrushTabLimEn" -SignalType "DO" -Access "All"

      -Name "A1BrushTable" -SignalType "AI" -Access "All"

--- Backups/Controlador_Pintura_v2/SYSPAR/PROC.cfg ---
PROC:CFG_1.0:6:0::
#
CONVEYOR:

      -name "CNV1" -sensor_type "CAN" -use_sensor "CAN1" -adjustment_speed 850\
      -min_dist -300 -max_dist 2500 -correction_vector_ramp_length 5
#
CONVEYOR_CAN_SENSOR:

      -name "CAN1" -eio_unit_name "Qtrack1" -connected_signal "c1Connected"\
      -position_signal "c1Position" -velocity_signal "c1Speed"\
      -null_speed_signal "c1NullSpeed" -wait_wobj_signal "c1WaitWObj"\
      -drop_wobj_signal "c1DropWObj" -data_timestamp "c1DTimestamp"\
      -rem_all_pobj_signal "c1RemAllPObj" -rem_one_pobj_signal "c1Rem1PObj"\
      -supervise_max_dist_off  -newobj_strobe "c1NewObjStrobe"\
      -encA_fault_signal "c1EncAFautlt" -dir_of_travel_signal "c1DirOfTravel"\
      -force_job_signal "c1ForceJob" -count_to_enc_strobe "c1CntToEncStr"\
      -pos_in_jobq_signal "c1PosInJobQ" -obj_in_queue_signal "c1ObjectsInQ"\
      -count_from_enc "c1CntFromEnc" -count_to_enc "c1CntToEnc"\
      -scale_enc_puls "c1ScaleEncPuls"
#
PW_SYSTEM:

      -name "PW_SYS" -pw_function "PW_FUNC"
#
PW_FUNCTION:

      -name "PW_FUNC" -do_repos_finished "ReposFinished"
#
PW_SERVICES_CONFIG:

      -Name "ProgramDirectory" -Value "HOME:/programs/"

      -Name "ProgramCache" -Value "False"

      -Name "LoadFailureModule" -Value ""

      -Name "ProgramStaticLoad" -Value "False"

      -Name "ProgramBackupSave" -Value "False"

      -Name "ProdLogDirectory" -Value "HOME:/logs"

      -Name "ProdLogFormat"\
      -Value "%D,Prog:%P,Mtrl:%M,Brush:%B,Usage:%C,CycleTime:%T"

      -Name "ProdLogSize" -Value "100000"

      -Name "JobQueueSize" -Value "10"

      -Name "JobQueueSave" -Value "False"

      -Name "JobQueueExpediteBegin" -Value "10001"

      -Name "JobQueueExpediteEnd" -Value "10016"

      -Name "ProgramIndexFile" -Value "HOME:/programs/segments.ndx"

      -Name "ExternalStart" -Value "False"

      -Name "JobQueueIgnoreMaterial" -Value "True"

      -Name "TipCleanModule" -Value "TipClean"

      -Name "TipCleanInterval" -Value "0"

      -Name "TipCleanModuleFile" -Value ""

      -Name "TipCleanIntervalFile" -Value ""

      -Name "AppCleanModule" -Value "AppClean"

      -Name "AppCleanInterval" -Value "0"

      -Name "AppCleanModuleFile" -Value ""

      -Name "AppCleanIntervalFile" -Value ""

      -Name "AppCleanHasPriority" -Value "False"

      -Name "BrushMapFormula" -Value "M"

      -Name "BrushMapFilter" -Value "999999"

      -Name "BrushMapZeroDefault" -Value "0"

      -Name "BrushTableDirectory" -Value "HOME:/ipsdata/node1/A1Brush/"

      -Name "HVAckSignal" -Value "HV_ILCK_ACK"

      -Name "HVAckDelay" -Value "200"

      -Name "A1EnableSignal" -Value "A1Enable"

      -Name "A1ErrorSignal" -Value "A1Error"

      -Name "A1BrushTabNdxSignal" -Value "A1BrushTabNdx"

      -Name "A1BrushTableSignal" -Value "A1BrushTable"

      -Name "A1BrushTabLimEnSignal" -Value "A1BrushTabLimEn"

      -Name "A1FluidAccuSignal" -Value "A1FluidAccu"

      -Name "A1HVEnSignal" -Value "A1HVEn"

      -Name "A1HVErrNoSignal" -Value "A1HVErrNo"

      -Name "A1BrushDevice" -Value "A1Brush"

      -Name "A1FluidEnSignal" -Value "A1FluidEn"

      -Name "A1NeedleEnSignal" -Value "A1NeedleEn"

      -Name "A1MaterialSignal" -Value "A1Material"

      -Name "BrushTrackSignal" -Value "A1Brush"

      -Name "BrushTrackDirectory" -Value "HOME:/btrack/"

      -Name "BrushTrackFormula" -Value "P"

      -Name "CmdLogDirectory" -Value "HOME:/logs"

      -Name "CmdLogSize" -Value "100000"

      -Name "RobotDataDirectory" -Value "HOME:/robdata/"

      -Name "ProgramAliasFile" -Value "HOME:/alias/program.map"

      -Name "MaterialAliasFile" -Value "HOME:/alias/material.map"

      -Name "OptionAliasFile" -Value "HOME:/alias/option.map"
#
PW_EVENT_HOOKS:

      -Routine "TipCleanPreMain" -Event "PRE_MAIN" -Priority 55

      -Routine "TipCleanPostMain" -Event "POST_MAIN" -Priority 75

      -Routine "ResetConvTime" -Event "PRE_MAIN" -Priority 60

      -Routine "PreMainPosMsg" -Event "PRE_MAIN" -Priority 80

      -Routine "PostMainPosMsg" -Event "POST_MAIN" -Priority 20

      -Routine "PreMainCustom" -Event "PRE_MAIN"

      -Routine "PostMainCustom" -Event "POST_MAIN"
#
PW_SIGNAL_OUT:

      -Status "Resource:Loop.InJob" -Signal "JobInProgress"

      -Status "Resource:Loop.InModule" -Signal "doInModule"

      -Status "Resource:Loop.ProgramLoaded" -Signal "ProgramLoaded"

      -Status "Resource:Queue.Empty" -Signal "doQueueEmpty"

      -Status "Resource:Queue.Inhibited" -Signal "doQueuePause"

      -Status "Resource:MCEngine.Suspended" -Signal "doMCSuspended"

      -Status "Resource:MCEngine.On" -Signal "MtrlChangeOn"

      -Status "Resource:MCLog.ErrorStatus" -Signal "MtrlSupplyError"

      -Status "Resource:Queue.Full" -Signal "doQueueFull"

      -Status "Resource:App.HVError" -Signal "HVError"

      -Status "Resource:Sup.PowerError" -Signal "PowerError"
